KUKA KRL program: TMatriz.src, TMatriz.dat

--- TMatriz.src ---
&ACCESS RV1
DEF TMatriz()
;FOLD PALLET 1
;FOLD Pallet 1 - Produto 9Aero
;FOLD LAYER 1: PLACE 1 ate 2
;FOLD PLACE 1
;FOLD PROPRIEDADES
MatrizPontos[Pallet_1,Prdt_9Aero,1].NumCaixas = 4
MatrizPontos[Pallet_1,Prdt_9Aero,1].PickOp = 3
MatrizPontos[Pallet_1,Prdt_9Aero,1].ConfGarraOp = 3
MatrizPontos[Pallet_1,Prdt_9Aero,1].FechaGarraOp = 0
MatrizPontos[Pallet_1,Prdt_9Aero,1].AbreGarraOp = 0
MatrizPontos[Pallet_1,Prdt_9Aero,1].SensoresCaixa = 123456
MatrizPontos[Pallet_1,Prdt_9Aero,1].TravaGarra = False
MatrizPontos[Pallet_1,Prdt_9Aero,1].SkipGoHome = False
MatrizPontos[Pallet_1,Prdt_9Aero,1].SkipSobeRelAtual = False
MatrizPontos[Pallet_1,Prdt_9Aero,1].XApp1Place=P1_9Aero_1_App1
MatrizPontos[Pallet_1,Prdt_9Aero,1].XApp2Place=P1_9Aero_1_App2
MatrizPontos[Pallet_1,Prdt_9Aero,1].XPlace=P1_9Aero_1_Place
;ENDFOLD
;FOLD OffsetPlace
MatrizPontos[Pallet_1,Prdt_9Aero,1].OffsetPlace.X=0
MatrizPontos[Pallet_1,Prdt_9Aero,1].OffsetPlace.Y=0
MatrizPontos[Pallet_1,Prdt_9Aero,1].OffsetPlace.Z=0
MatrizPontos[Pallet_1,Prdt_9Aero,1].OffsetPlace.A=0
MatrizPontos[Pallet_1,Prdt_9Aero,1].OffsetPlace.B=0
MatrizPontos[Pallet_1,Prdt_9Aero,1].OffsetPlace.C=0
;ENDFOLD
;ENDFOLD

;FOLD PLACE 2
;FOLD PROPRIEDADES
MatrizPontos[Pallet_1,Prdt_9Aero,2].NumCaixas = 4
MatrizPontos[Pallet_1,Prdt_9Aero,2].PickOp = 3
MatrizPontos[Pallet_1,Prdt_9Aero,2].ConfGarraOp = 3
MatrizPontos[Pallet_1,Prdt_9Aero,2].FechaGarraOp = 0
MatrizPontos[Pallet_1,Prdt_9Aero,2].AbreGarraOp = 0
MatrizPontos[Pallet_1,Prdt_9Aero,2].SensoresCaixa = 123456
MatrizPontos[Pallet_1,Prdt_9Aero,2].TravaGarra = False
MatrizPontos[Pallet_1,Prdt_9Aero,2].SkipGoHome = False
MatrizPontos[Pallet_1,Prdt_9Aero,2].SkipSobeRelAtual = False
MatrizPontos[Pallet_1,Prdt_9Aero,2].XApp1Place=P1_9Aero_2_App1
MatrizPontos[Pallet_1,Prdt_9Aero,2].XApp2Place=P1_9Aero_2_App2
MatrizPontos[Pallet_1,Prdt_9Aero,2].XPlace=P1_9Aero_2_Place
;ENDFOLD
;FOLD OffsetPlace
MatrizPontos[Pallet_1,Prdt_9Aero,2].OffsetPlace.X=0
MatrizPontos[Pallet_1,Prdt_9Aero,2].OffsetPlace.Y=0
MatrizPontos[Pallet_1,Prdt_9Aero,2].OffsetPlace.Z=0
MatrizPontos[Pallet_1,Prdt_9Aero,2].OffsetPlace.A=0
MatrizPontos[Pallet_1,Prdt_9Aero,2].OffsetPlace.B=0
MatrizPontos[Pallet_1,Prdt_9Aero,2].OffsetPlace.C=0
;ENDFOLD
;ENDFOLD

;ENDFOLD
;ENDFOLD

;FOLD Pallet 1 - Produto 5Aero
;FOLD LAYER 1: PLACE 1 ate 3
;FOLD PLACE 1
;FOLD PROPRIEDADES
MatrizPontos[Pallet_1,Prdt_5Aero,1].NumCaixas = 3
MatrizPontos[Pallet_1,Prdt_5Aero,1].PickOp = 1
MatrizPontos[Pallet_1,Prdt_5Aero,1].ConfGarraOp = 0
MatrizPontos[Pallet_1,Prdt_5Aero,1].FechaGarraOp = 0
MatrizPontos[Pallet_1,Prdt_5Aero,1].AbreGarraOp = 0
MatrizPontos[Pallet_1,Prdt_5Aero,1].SensoresCaixa = 12345
MatrizPontos[Pallet_1,Prdt_5Aero,1].TravaGarra = False
MatrizPontos[Pallet_1,Prdt_5Aero,1].SkipGoHome = False
MatrizPontos[Pallet_1,Prdt_5Aero,1].SkipSobeRelAtual = False
MatrizPontos[Pallet_1,Prdt_5Aero,1].XApp1Place=P1_5Aero_1_App1
MatrizPontos[Pallet_1,Prdt_5Aero,1].XApp2Place=P1_5Aero_1_App2
MatrizPontos[Pallet_1,Prdt_5Aero,1].XPlace=P1_5Aero_1_Place
;ENDFOLD
;FOLD OffsetPlace
MatrizPontos[Pallet_1,Prdt_5Aero,1].OffsetPlace.X=0
MatrizPontos[Pallet_1,Prdt_5Aero,1].OffsetPlace.Y=0
MatrizPontos[Pallet_1,Prdt_5Aero,1].OffsetPlace.Z=0
MatrizPontos[Pallet_1,Prdt_5Aero,1].OffsetPlace.A=0
MatrizPontos[Pallet_1,Prdt_5Aero,1].OffsetPlace.B=0
MatrizPontos[Pallet_1,Prdt_5Aero,1].OffsetPlace.C=0
;ENDFOLD
;ENDFOLD

;FOLD PLACE 2
;FOLD PROPRIEDADES
MatrizPontos[Pallet_1,Prdt_5Aero,2].NumCaixas = 3
MatrizPontos[Pallet_1,Prdt_5Aero,2].PickOp = 1
MatrizPontos[Pallet_1,Prdt_5Aero,2].ConfGarraOp = 0
MatrizPontos[Pallet_1,Prdt_5Aero,2].FechaGarraOp = 0
MatrizPontos[Pallet_1,Prdt_5Aero,2].AbreGarraOp = 0
MatrizPontos[Pallet_1,Prdt_5Aero,2].SensoresCaixa = 12345
MatrizPontos[Pallet_1,Prdt_5Aero,2].TravaGarra = False
MatrizPontos[Pallet_1,Prdt_5Aero,2].SkipGoHome = False
MatrizPontos[Pallet_1,Prdt_5Aero,2].SkipSobeRelAtual = False
MatrizPontos[Pallet_1,Prdt_5Aero,2].XApp1Place=P1_5Aero_2_App1
MatrizPontos[Pallet_1,Prdt_5Aero,2].XApp2Place=P1_5Aero_2_App2
MatrizPontos[Pallet_1,Prdt_5Aero,2].XPlace=P1_5Aero_2_Place
;ENDFOLD
;FOLD OffsetPlace
MatrizPontos[Pallet_1,Prdt_5Aero,2].OffsetPlace.X=0
MatrizPontos[Pallet_1,Prdt_5Aero,2].OffsetPlace.Y=0
MatrizPontos[Pallet_1,Prdt_5Aero,2].OffsetPlace.Z=0
MatrizPontos[Pallet_1,Prdt_5Aero,2].OffsetPlace.A=0
MatrizPontos[Pallet_1,Prdt_5Aero,2].OffsetPlace.B=0
MatrizPontos[Pallet_1,Prdt_5Aero,2].OffsetPlace.C=0
;ENDFOLD
;ENDFOLD

;FOLD PLACE 3
;FOLD PROPRIEDADES
MatrizPontos[Pallet_1,Prdt_5Aero,3].NumCaixas = 3
MatrizPontos[Pallet_1,Prdt_5Aero,3].PickOp = 1
MatrizPontos[Pallet_1,Prdt_5Aero,3].ConfGarraOp = 0
MatrizPontos[Pallet_1,Prdt_5Aero,3].FechaGarraOp = 0
MatrizPontos[Pallet_1,Prdt_5Aero,3].AbreGarraOp = 0
MatrizPontos[Pallet_1,Prdt_5Aero,3].SensoresCaixa = 12345
MatrizPontos[Pallet_1,Prdt_5Aero,3].TravaGarra = False
MatrizPontos[Pallet_1,Prdt_5Aero,3].SkipGoHome = False
MatrizPontos[Pallet_1,Prdt_5Aero,3].SkipSobeRelAtual = False
MatrizPontos[Pallet_1,Prdt_5Aero,3].XApp1Place=P1_5Aero_3_App1
MatrizPontos[Pallet_1,Prdt_5Aero,3].XApp2Place=P1_5Aero_3_App2
MatrizPontos[Pallet_1,Prdt_5Aero,3].XPlace=P1_5Aero_3_Place
;ENDFOLD
;FOLD OffsetPlace
MatrizPontos[Pallet_1,Prdt_5Aero,3].OffsetPlace.X=0
MatrizPontos[Pallet_1,Prdt_5Aero,3].OffsetPlace.Y=0
MatrizPontos[Pallet_1,Prdt_5Aero,3].OffsetPlace.Z=0
MatrizPontos[Pallet_1,Prdt_5Aero,3].OffsetPlace.A=0
MatrizPontos[Pallet_1,Prdt_5Aero,3].OffsetPlace.B=0
MatrizPontos[Pallet_1,Prdt_5Aero,3].OffsetPlace.C=0
;ENDFOLD
;ENDFOLD

;ENDFOLD
;ENDFOLD

;FOLD Pallet 1 - Produto 2Aero
;FOLD LAYER 1: PLACE 1 ate 3
;FOLD PLACE 1
;FOLD PROPRIEDADES
MatrizPontos[Pallet_1,Prdt_2Aero,1].NumCaixas = 4
MatrizPontos[Pallet_1,Prdt_2Aero,1].PickOp = 1
MatrizPontos[Pallet_1,Prdt_2Aero,1].ConfGarraOp = 0
MatrizPontos[Pallet_1,Prdt_2Aero,1].FechaGarraOp = 0
MatrizPontos[Pallet_1,Prdt_2Aero,1].AbreGarraOp = 0
MatrizPontos[Pallet_1,Prdt_2Aero,1].SensoresCaixa = 123456
MatrizPontos[Pallet_1,Prdt_2Aero,1].TravaGarra = False
MatrizPontos[Pallet_1,Prdt_2Aero,1].SkipGoHome = False
MatrizPontos[Pallet_1,Prdt_2Aero,1].SkipSobeRelAtual = False
MatrizPontos[Pallet_1,Prdt_2Aero,1].XApp1Place=P1_2Aero_1_App1
MatrizPontos[Pallet_1,Prdt_2Aero,1].XApp2Place=P1_2Aero_1_App2
MatrizPontos[Pallet_1,Prdt_2Aero,1].XPlace=P1_2Aero_1_Place
;ENDFOLD
;FOLD OffsetPlace
MatrizPontos[Pallet_1,Prdt_2Aero,1].OffsetPlace.X=0
MatrizPontos[Pallet_1,Prdt_2Aero,1].OffsetPlace.Y=0
MatrizPontos[Pallet_1,Prdt_2Aero,1].OffsetPlace.Z=0
MatrizPontos[Pallet_1,Prdt_2Aero,1].OffsetPlace.A=0
MatrizPontos[Pallet_1,Prdt_2Aero,1].OffsetPlace.B=0
MatrizPontos[Pallet_1,Prdt_2Aero,1].OffsetPlace.C=0
;ENDFOLD
;ENDFOLD

;FOLD PLACE 2
;FOLD PROPRIEDADES
MatrizPontos[Pallet_1,Prdt_2Aero,2].NumCaixas = 4
MatrizPontos[Pallet_1,Prdt_2Aero,2].PickOp = 1
MatrizPontos[Pallet_1,Prdt_2Aero,2].ConfGarraOp = 0
MatrizPontos[Pallet_1,Prdt_2Aero,2].FechaGarraOp = 0
MatrizPontos[Pallet_1,Prdt_2Aero,2].AbreGarraOp = 0
MatrizPontos[Pallet_1,Prdt_2Aero,2].SensoresCaixa = 123456
MatrizPontos[Pallet_1,Prdt_2Aero,2].TravaGarra = False
MatrizPontos[Pallet_1,Prdt_2Aero,2].SkipGoHome = False
MatrizPontos[Pallet_1,Prdt_2Aero,2].SkipSobeRelAtual = False
MatrizPontos[Pallet_1,Prdt_2Aero,2].XApp1Place=P1_2Aero_2_App1
MatrizPontos[Pallet_1,Prdt_2Aero,2].XApp2Place=P1_2Aero_2_App2
MatrizPontos[Pallet_1,Prdt_2Aero,2].XPlace=P1_2Aero_2_Place
;ENDFOLD
;FOLD OffsetPlace
MatrizPontos[Pallet_1,Prdt_2Aero,2].OffsetPlace.X=0
MatrizPontos[Pallet_1,Prdt_2Aero,2].OffsetPlace.Y=0
MatrizPontos[Pallet_1,Prdt_2Aero,2].OffsetPlace.Z=0
MatrizPontos[Pallet_1,Prdt_2Aero,2].OffsetPlace.A=0
MatrizPontos[Pallet_1,Prdt_2Aero,2].OffsetPlace.B=0
MatrizPontos[Pallet_1,Prdt_2Aero,2].OffsetPlace.C=0
;ENDFOLD
;ENDFOLD

;FOLD PLACE 3
;FOLD PROPRIEDADES
MatrizPontos[Pallet_1,Prdt_2Aero,3].NumCaixas = 4
MatrizPontos[Pallet_1,Prdt_2Aero,3].PickOp = 1
MatrizPontos[Pallet_1,Prdt_2Aero,3].ConfGarraOp = 0
MatrizPontos[Pallet_1,Prdt_2Aero,3].FechaGarraOp = 0
MatrizPontos[Pallet_1,Prdt_2Aero,3].AbreGarraOp = 0
MatrizPontos[Pallet_1,Prdt_2Aero,3].SensoresCaixa = 123456
MatrizPontos[Pallet_1,Prdt_2Aero,3].TravaGarra = False
MatrizPontos[Pallet_1,Prdt_2Aero,3].SkipGoHome = False
MatrizPontos[Pallet_1,Prdt_2Aero,3].SkipSobeRelAtual = False
MatrizPontos[Pallet_1,Prdt_2Aero,3].XApp1Place=P1_2Aero_3_App1
MatrizPontos[Pallet_1,Prdt_2Aero,3].XApp2Place=P1_2Aero_3_App2
MatrizPontos[Pallet_1,Prdt_2Aero,3].XPlace=P1_2Aero_3_Place
;ENDFOLD
;FOLD OffsetPlace
MatrizPontos[Pallet_1,Prdt_2Aero,3].OffsetPlace.X=0
MatrizPontos[Pallet_1,Prdt_2Aero,3].OffsetPlace.Y=0
MatrizPontos[Pallet_1,Prdt_2Aero,3].OffsetPlace.Z=0
MatrizPontos[Pallet_1,Prdt_2Aero,3].OffsetPlace.A=0
MatrizPontos[Pallet_1,Prdt_2Aero,3].OffsetPlace.B=0
MatrizPontos[Pallet_1,Prdt_2Aero,3].OffsetPlace.C=0
;ENDFOLD
;ENDFOLD

;ENDFOLD
;ENDFOLD

;FOLD Pallet 1 - Produto 11CoffeCrisp
;FOLD LAYER 1: PLACE 1 ate 3
;FOLD PLACE 1
;FOLD PROPRIEDADES
MatrizPontos[Pallet_1,Prdt_11CoffeCrisp,1].NumCaixas = 3
MatrizPontos[Pallet_1,Prdt_11CoffeCrisp,1].PickOp = 1
MatrizPontos[Pallet_1,Prdt_11CoffeCrisp,1].ConfGarraOp = 0
MatrizPontos[Pallet_1,Prdt_11CoffeCrisp,1].FechaGarraOp = 0
MatrizPontos[Pallet_1,Prdt_11CoffeCrisp,1].AbreGarraOp = 0
MatrizPontos[Pallet_1,Prdt_11CoffeCrisp,1].SensoresCaixa = 12345
MatrizPontos[Pallet_1,Prdt_11CoffeCrisp,1].TravaGarra = False
MatrizPontos[Pallet_1,Prdt_11CoffeCrisp,1].SkipGoHome = False
MatrizPontos[Pallet_1,Prdt_11CoffeCrisp,1].SkipSobeRelAtual = False
MatrizPontos[Pallet_1,Prdt_11CoffeCrisp,1].XApp1Place=P1_11CoffeCrisp_1_App1
MatrizPontos[Pallet_1,Prdt_11CoffeCrisp,1].XApp2Place=P1_11CoffeCrisp_1_App2
MatrizPontos[Pallet_1,Prdt_11CoffeCrisp,1].XPlace=P1_11CoffeCrisp_1_Place
;ENDFOLD
;FOLD OffsetPlace
MatrizPontos[Pallet_1,Prdt_11CoffeCrisp,1].OffsetPlace.X=0
MatrizPontos[Pallet_1,Prdt_11CoffeCrisp,1].OffsetPlace.Y=0
MatrizPontos[Pallet_1,Prdt_11CoffeCrisp,1].OffsetPlace.Z=0
MatrizPontos[Pallet_1,Prdt_11CoffeCrisp,1].OffsetPlace.A=0
MatrizPontos[Pallet_1,Prdt_11CoffeCrisp,1].OffsetPlace.B=0
MatrizPontos[Pallet_1,Prdt_11CoffeCrisp,1].OffsetPlace.C=0
;ENDFOLD
;ENDFOLD

;FOLD PLACE 2
;FOLD PROPRIEDADES
MatrizPontos[Pallet_1,Prdt_11CoffeCrisp,2].NumCaixas = 3
MatrizPontos[Pallet_1,Prdt_11CoffeCrisp,2].PickOp = 1
MatrizPontos[Pallet_1,Prdt_11CoffeCrisp,2].ConfGarraOp = 0
MatrizPontos[Pallet_1,Prdt_11CoffeCrisp,2].FechaGarraOp = 0
MatrizPontos[Pallet_1,Prdt_11CoffeCrisp,2].AbreGarraOp = 0
MatrizPontos[Pallet_1,Prdt_11CoffeCrisp,2].SensoresCaixa = 12345
MatrizPontos[Pallet_1,Prdt_11CoffeCrisp,2].TravaGarra = False
MatrizPontos[Pallet_1,Prdt_11CoffeCrisp,2].SkipGoHome = False
MatrizPontos[Pallet_1,Prdt_11CoffeCrisp,2].SkipSobeRelAtual = False
MatrizPontos[Pallet_1,Prdt_11CoffeCrisp,2].XApp1Place=P1_11CoffeCrisp_2_App1
MatrizPontos[Pallet_1,Prdt_11CoffeCrisp,2].XApp2Place=P1_11CoffeCrisp_2_App2
MatrizPontos[Pallet_1,Prdt_11CoffeCrisp,2].XPlace=P1_11CoffeCrisp_2_Place
;ENDFOLD
;FOLD OffsetPlace
MatrizPontos[Pallet_1,Prdt_11CoffeCrisp,2].OffsetPlace.X=0
MatrizPontos[Pallet_1,Prdt_11CoffeCrisp,2].OffsetPlace.Y=0
MatrizPontos[Pallet_1,Prdt_11CoffeCrisp,2].OffsetPlace.Z=0
MatrizPontos[Pallet_1,Prdt_11CoffeCrisp,2].OffsetPlace.A=0
MatrizPontos[Pallet_1,Prdt_11CoffeCrisp,2].OffsetPlace.B=0
MatrizPontos[Pallet_1,Prdt_11CoffeCrisp,2].OffsetPlace.C=0
;ENDFOLD
;ENDFOLD

;FOLD PLACE 3
;FOLD PROPRIEDADES
MatrizPontos[Pallet_1,Prdt_11CoffeCrisp,3].NumCaixas = 3
MatrizPontos[Pallet_1,Prdt_11CoffeCrisp,3].PickOp = 1
MatrizPontos[Pallet_1,Prdt_11CoffeCrisp,3].ConfGarraOp = 0
MatrizPontos[Pallet_1,Prdt_11CoffeCrisp,3].FechaGarraOp = 0
MatrizPontos[Pallet_1,Prdt_11CoffeCrisp,3].AbreGarraOp = 0
MatrizPontos[Pallet_1,Prdt_11CoffeCrisp,3].SensoresCaixa = 12345
MatrizPontos[Pallet_1,Prdt_11CoffeCrisp,3].TravaGarra = False
MatrizPontos[Pallet_1,Prdt_11CoffeCrisp,3].SkipGoHome = False
MatrizPontos[Pallet_1,Prdt_11CoffeCrisp,3].SkipSobeRelAtual = False
MatrizPontos[Pallet_1,Prdt_11CoffeCrisp,3].XApp1Place=P1_11CoffeCrisp_3_App1
MatrizPontos[Pallet_1,Prdt_11CoffeCrisp,3].XApp2Place=P1_11CoffeCrisp_3_App2
MatrizPontos[Pallet_1,Prdt_11CoffeCrisp,3].XPlace=P1_11CoffeCrisp_3_Place
;ENDFOLD
;FOLD OffsetPlace
MatrizPontos[Pallet_1,Prdt_11CoffeCrisp,3].OffsetPlace.X=0
MatrizPontos[Pallet_1,Prdt_11CoffeCrisp,3].OffsetPlace.Y=0
MatrizPontos[Pallet_1,Prdt_11CoffeCrisp,3].OffsetPlace.Z=0
MatrizPontos[Pallet_1,Prdt_11CoffeCrisp,3].OffsetPlace.A=0
MatrizPontos[Pallet_1,Prdt_11CoffeCrisp,3].OffsetPlace.B=0
MatrizPontos[Pallet_1,Prdt_11CoffeCrisp,3].OffsetPlace.C=0
;ENDFOLD
;ENDFOLD

;ENDFOLD
;ENDFOLD

;FOLD Pallet 1 - Produto 17KitKat
;FOLD LAYER 1: PLACE 1 ate 4
;FOLD PLACE 1
;FOLD PROPRIEDADES
MatrizPontos[Pallet_1,Prdt_17KitKat,1].NumCaixas = 3
MatrizPontos[Pallet_1,Prdt_17KitKat,1].PickOp = 1
MatrizPontos[Pallet_1,Prdt_17KitKat,1].ConfGarraOp = 0
MatrizPontos[Pallet_1,Prdt_17KitKat,1].FechaGarraOp = 0
MatrizPontos[Pallet_1,Prdt_17KitKat,1].AbreGarraOp = 0
MatrizPontos[Pallet_1,Prdt_17KitKat,1].SensoresCaixa = 1234
MatrizPontos[Pallet_1,Prdt_17KitKat,1].TravaGarra = False
MatrizPontos[Pallet_1,Prdt_17KitKat,1].SkipGoHome = False
MatrizPontos[Pallet_1,Prdt_17KitKat,1].SkipSobeRelAtual = False
MatrizPontos[Pallet_1,Prdt_17KitKat,1].XApp1Place=P1_17KitKat_1_App1
MatrizPontos[Pallet_1,Prdt_17KitKat,1].XApp2Place=P1_17KitKat_1_App2
MatrizPontos[Pallet_1,Prdt_17KitKat,1].XPlace=P1_17KitKat_1_Place
;ENDFOLD
;FOLD OffsetPlace
MatrizPontos[Pallet_1,Prdt_17KitKat,1].OffsetPlace.X=0
MatrizPontos[Pallet_1,Prdt_17KitKat,1].OffsetPlace.Y=0
MatrizPontos[Pallet_1,Prdt_17KitKat,1].OffsetPlace.Z=0
MatrizPontos[Pallet_1,Prdt_17KitKat,1].OffsetPlace.A=0
MatrizPontos[Pallet_1,Prdt_17KitKat,1].OffsetPlace.B=0
MatrizPontos[Pallet_1,Prdt_17KitKat,1].OffsetPlace.C=0
;ENDFOLD
;ENDFOLD

;FOLD PLACE 2
;FOLD PROPRIEDADES
MatrizPontos[Pallet_1,Prdt_17KitKat,2].NumCaixas = 3
MatrizPontos[Pallet_1,Prdt_17KitKat,2].PickOp = 1
MatrizPontos[Pallet_1,Prdt_17KitKat,2].ConfGarraOp = 0
MatrizPontos[Pallet_1,Prdt_17KitKat,2].FechaGarraOp = 0
MatrizPontos[Pallet_1,Prdt_17KitKat,2].AbreGarraOp = 0
MatrizPontos[Pallet_1,Prdt_17KitKat,2].SensoresCaixa = 1234
MatrizPontos[Pallet_1,Prdt_17KitKat,2].TravaGarra = False
MatrizPontos[Pallet_1,Prdt_17KitKat,2].SkipGoHome = False
MatrizPontos[Pallet_1,Prdt_17KitKat,2].SkipSobeRelAtual = False
MatrizPontos[Pallet_1,Prdt_17KitKat,2].XApp1Place=P1_17KitKat_2_App1
MatrizPontos[Pallet_1,Prdt_17KitKat,2].XApp2Place=P1_17KitKat_2_App2
MatrizPontos[Pallet_1,Prdt_17KitKat,2].XPlace=P1_17KitKat_2_Place
;ENDFOLD
;FOLD OffsetPlace
MatrizPontos[Pallet_1,Prdt_17KitKat,2].OffsetPlace.X=0
MatrizPontos[Pallet_1,Prdt_17KitKat,2].OffsetPlace.Y=0
MatrizPontos[Pallet_1,Prdt_17KitKat,2].OffsetPlace.Z=0
MatrizPontos[Pallet_1,Prdt_17KitKat,2].OffsetPlace.A=0
MatrizPontos[Pallet_1,Prdt_17KitKat,2].OffsetPlace.B=0
MatrizPontos[Pallet_1,Prdt_17KitKat,2].OffsetPlace.C=0
;ENDFOLD
;ENDFOLD

;FOLD PLACE 3
;FOLD PROPRIEDADES
MatrizPontos[Pallet_1,Prdt_17KitKat,3].NumCaixas = 3
MatrizPontos[Pallet_1,Prdt_17KitKat,3].PickOp = 1
MatrizPontos[Pallet_1,Prdt_17KitKat,3].ConfGarraOp = 0
MatrizPontos[Pallet_1,Prdt_17KitKat,3].FechaGarraOp = 0
MatrizPontos[Pallet_1,Prdt_17KitKat,3].AbreGarraOp = 0
MatrizPontos[Pallet_1,Prdt_17KitKat,3].SensoresCaixa = 1234
MatrizPontos[Pallet_1,Prdt_17KitKat,3].TravaGarra = False
MatrizPontos[Pallet_1,Prdt_17KitKat,3].SkipGoHome = False
MatrizPontos[Pallet_1,Prdt_17KitKat,3].SkipSobeRelAtual = False
MatrizPontos[Pallet_1,Prdt_17KitKat,3].XApp1Place=P1_17KitKat_3_App1
MatrizPontos[Pallet_1,Prdt_17KitKat,3].XApp2Place=P1_17KitKat_3_App2
MatrizPontos[Pallet_1,Prdt_17KitKat,3].XPlace=P1_17KitKat_3_Place
;ENDFOLD
;FOLD OffsetPlace
MatrizPontos[Pallet_1,Prdt_17KitKat,3].OffsetPlace.X=0
MatrizPontos[Pallet_1,Prdt_17KitKat,3].OffsetPlace.Y=0
MatrizPontos[Pallet_1,Prdt_17KitKat,3].OffsetPlace.Z=0
MatrizPontos[Pallet_1,Prdt_17KitKat,3].OffsetPlace.A=0
MatrizPontos[Pallet_1,Prdt_17KitKat,3].OffsetPlace.B=0
MatrizPontos[Pallet_1,Prdt_17KitKat,3].OffsetPlace.C=0
;ENDFOLD
;ENDFOLD

;FOLD PLACE 4
;FOLD PROPRIEDADES
MatrizPontos[Pallet_1,Prdt_17KitKat,4].NumCaixas = 3
MatrizPontos[Pallet_1,Prdt_17KitKat,4].PickOp = 1
MatrizPontos[Pallet_1,Prdt_17KitKat,4].ConfGarraOp = 0
MatrizPontos[Pallet_1,Prdt_17KitKat,4].FechaGarraOp = 0
MatrizPontos[Pallet_1,Prdt_17KitKat,4].AbreGarraOp = 0
MatrizPontos[Pallet_1,Prdt_17KitKat,4].SensoresCaixa = 1234
MatrizPontos[Pallet_1,Prdt_17KitKat,4].TravaGarra = False
MatrizPontos[Pallet_1,Prdt_17KitKat,4].SkipGoHome = False
MatrizPontos[Pallet_1,Prdt_17KitKat,4].SkipSobeRelAtual = False
MatrizPontos[Pallet_1,Prdt_17KitKat,4].XApp1Place=P1_17KitKat_4_App1
MatrizPontos[Pallet_1,Prdt_17KitKat,4].XApp2Place=P1_17KitKat_4_App2
MatrizPontos[Pallet_1,Prdt_17KitKat,4].XPlace=P1_17KitKat_4_Place
;ENDFOLD
;FOLD OffsetPlace
MatrizPontos[Pallet_1,Prdt_17KitKat,4].OffsetPlace.X=0
MatrizPontos[Pallet_1,Prdt_17KitKat,4].OffsetPlace.Y=0
MatrizPontos[Pallet_1,Prdt_17KitKat,4].OffsetPlace.Z=0
MatrizPontos[Pallet_1,Prdt_17KitKat,4].OffsetPlace.A=0
MatrizPontos[Pallet_1,Prdt_17KitKat,4].OffsetPlace.B=0
MatrizPontos[Pallet_1,Prdt_17KitKat,4].OffsetPlace.C=0
;ENDFOLD
;ENDFOLD

;ENDFOLD
;ENDFOLD

;FOLD Pallet 1 - Produto 19KitKat
;FOLD LAYER 1: PLACE 1 ate 6
;FOLD PLACE 1
;FOLD PROPRIEDADES
MatrizPontos[Pallet_1,Prdt_19KitKat,1].NumCaixas = 1
MatrizPontos[Pallet_1,Prdt_19KitKat,1].PickOp = 6
MatrizPontos[Pallet_1,Prdt_19KitKat,1].ConfGarraOp = 0
MatrizPontos[Pallet_1,Prdt_19KitKat,1].FechaGarraOp = 0
MatrizPontos[Pallet_1,Prdt_19KitKat,1].AbreGarraOp = 0
MatrizPontos[Pallet_1,Prdt_19KitKat,1].SensoresCaixa = 6
MatrizPontos[Pallet_1,Prdt_19KitKat,1].TravaGarra = False
MatrizPontos[Pallet_1,Prdt_19KitKat,1].SkipGoHome = False
MatrizPontos[Pallet_1,Prdt_19KitKat,1].SkipSobeRelAtual = False
MatrizPontos[Pallet_1,Prdt_19KitKat,1].XApp1Place=P1_19KitKat_1_App1
MatrizPontos[Pallet_1,Prdt_19KitKat,1].XApp2Place=P1_19KitKat_1_App2
MatrizPontos[Pallet_1,Prdt_19KitKat,1].XPlace=P1_19KitKat_1_Place
;ENDFOLD
;FOLD OffsetPlace
MatrizPontos[Pallet_1,Prdt_19KitKat,1].OffsetPlace.X=0
MatrizPontos[Pallet_1,Prdt_19KitKat,1].OffsetPlace.Y=0
MatrizPontos[Pallet_1,Prdt_19KitKat,1].OffsetPlace.Z=0
MatrizPontos[Pallet_1,Prdt_19KitKat,1].OffsetPlace.A=0
MatrizPontos[Pallet_1,Prdt_19KitKat,1].OffsetPlace.B=0
MatrizPontos[Pallet_1,Prdt_19KitKat,1].OffsetPlace.C=0
;ENDFOLD
;ENDFOLD

;FOLD PLACE 2
;FOLD PROPRIEDADES
MatrizPontos[Pallet_1,Prdt_19KitKat,2].NumCaixas = 1
MatrizPontos[Pallet_1,Prdt_19KitKat,2].PickOp = 6
MatrizPontos[Pallet_1,Prdt_19KitKat,2].ConfGarraOp = 0
MatrizPontos[Pallet_1,Prdt_19KitKat,2].FechaGarraOp = 0
MatrizPontos[Pallet_1,Prdt_19KitKat,2].AbreGarraOp = 0
MatrizPontos[Pallet_1,Prdt_19KitKat,2].SensoresCaixa = 6
MatrizPontos[Pallet_1,Prdt_19KitKat,2].TravaGarra = False
MatrizPontos[Pallet_1,Prdt_19KitKat,2].SkipGoHome = False
MatrizPontos[Pallet_1,Prdt_19KitKat,2].SkipSobeRelAtual = False
MatrizPontos[Pallet_1,Prdt_19KitKat,2].XApp1Place=P1_19KitKat_2_App1
MatrizPontos[Pallet_1,Prdt_19KitKat,2].XApp2Place=P1_19KitKat_2_App2
MatrizPontos[Pallet_1,Prdt_19KitKat,2].XPlace=P1_19KitKat_2_Place
;ENDFOLD
;FOLD OffsetPlace
MatrizPontos[Pallet_1,Prdt_19KitKat,2].OffsetPlace.X=0
MatrizPontos[Pallet_1,Prdt_19KitKat,2].OffsetPlace.Y=0
MatrizPontos[Pallet_1,Prdt_19KitKat,2].OffsetPlace.Z=0
MatrizPontos[Pallet_1,Prdt_19KitKat,2].OffsetPlace.A=0
MatrizPontos[Pallet_1,Prdt_19KitKat,2].OffsetPlace.B=0
MatrizPontos[Pallet_1,Prdt_19KitKat,2].OffsetPlace.C=0
;ENDFOLD
;ENDFOLD

;FOLD PLACE 3
;FOLD PROPRIEDADES
MatrizPontos[Pallet_1,Prdt_19KitKat,3].NumCaixas = 1
MatrizPontos[Pallet_1,Prdt_19KitKat,3].PickOp = 6
MatrizPontos[Pallet_1,Prdt_19KitKat,3].ConfGarraOp = 0
MatrizPontos[Pallet_1,Prdt_19KitKat,3].FechaGarraOp = 0
MatrizPontos[Pallet_1,Prdt_19KitKat,3].AbreGarraOp = 0
MatrizPontos[Pallet_1,Prdt_19KitKat,3].SensoresCaixa = 6
MatrizPontos[Pallet_1,Prdt_19KitKat,3].TravaGarra = False
MatrizPontos[Pallet_1,Prdt_19KitKat,3].SkipGoHome = False
MatrizPontos[Pallet_1,Prdt_19KitKat,3].SkipSobeRelAtual = False
MatrizPontos[Pallet_1,Prdt_19KitKat,3].XApp1Place=P1_19KitKat_3_App1
MatrizPontos[Pallet_1,Prdt_19KitKat,3].XApp2Place=P1_19KitKat_3_App2
MatrizPontos[Pallet_1,Prdt_19KitKat,3].XPlace=P1_19KitKat_3_Place
;ENDFOLD
;FOLD OffsetPlace
MatrizPontos[Pallet_1,Prdt_19KitKat,3].OffsetPlace.X=0
MatrizPontos[Pallet_1,Prdt_19KitKat,3].OffsetPlace.Y=0
MatrizPontos[Pallet_1,Prdt_19KitKat,3].OffsetPlace.Z=0
MatrizPontos[Pallet_1,Prdt_19KitKat,3].OffsetPlace.A=0
MatrizPontos[Pallet_1,Prdt_19KitKat,3].OffsetPlace.B=0
MatrizPontos[Pallet_1,Prdt_19KitKat,3].OffsetPlace.C=0
;ENDFOLD
;ENDFOLD

;FOLD PLACE 4
;FOLD PROPRIEDADES
MatrizPontos[Pallet_1,Prdt_19KitKat,4].NumCaixas = 4
MatrizPontos[Pallet_1,Prdt_19KitKat,4].PickOp = 1
MatrizPontos[Pallet_1,Prdt_19KitKat,4].ConfGarraOp = 0
MatrizPontos[Pallet_1,Prdt_19KitKat,4].FechaGarraOp = 0
MatrizPontos[Pallet_1,Prdt_19KitKat,4].AbreGarraOp = 0
MatrizPontos[Pallet_1,Prdt_19KitKat,4].SensoresCaixa = 12345
MatrizPontos[Pallet_1,Prdt_19KitKat,4].TravaGarra = False
MatrizPontos[Pallet_1,Prdt_19KitKat,4].SkipGoHome = False
MatrizPontos[Pallet_1,Prdt_19KitKat,4].SkipSobeRelAtual = False
MatrizPontos[Pallet_1,Prdt_19KitKat,4].XApp1Place=P1_19KitKat_4_App1
MatrizPontos[Pallet_1,Prdt_19KitKat,4].XApp2Place=P1_19KitKat_4_App2
MatrizPontos[Pallet_1,Prdt_19KitKat,4].XPlace=P1_19KitKat_4_Place
;ENDFOLD
;FOLD OffsetPlace
MatrizPontos[Pallet_1,Prdt_19KitKat,4].OffsetPlace.X=0
MatrizPontos[Pallet_1,Prdt_19KitKat,4].OffsetPlace.Y=0
MatrizPontos[Pallet_1,Prdt_19KitKat,4].OffsetPlace.Z=0
MatrizPontos[Pallet_1,Prdt_19KitKat,4].OffsetPlace.A=0
MatrizPontos[Pallet_1,Prdt_19KitKat,4].OffsetPlace.B=0
MatrizPontos[Pallet_1,Prdt_19KitKat,4].OffsetPlace.C=0
;ENDFOLD
;ENDFOLD

;FOLD PLACE 5
;FOLD PROPRIEDADES
MatrizPontos[Pallet_1,Prdt_19KitKat,5].NumCaixas = 4
MatrizPontos[Pallet_1,Prdt_19KitKat,5].PickOp = 1
MatrizPontos[Pallet_1,Prdt_19KitKat,5].ConfGarraOp = 0
MatrizPontos[Pallet_1,Prdt_19KitKat,5].FechaGarraOp = 0
MatrizPontos[Pallet_1,Prdt_19KitKat,5].AbreGarraOp = 0
MatrizPontos[Pallet_1,Prdt_19KitKat,5].SensoresCaixa = 12345
MatrizPontos[Pallet_1,Prdt_19KitKat,5].TravaGarra = False
MatrizPontos[Pallet_1,Prdt_19KitKat,5].SkipGoHome = False
MatrizPontos[Pallet_1,Prdt_19KitKat,5].SkipSobeRelAtual = False
MatrizPontos[Pallet_1,Prdt_19KitKat,5].XApp1Place=P1_19KitKat_5_App1
MatrizPontos[Pallet_1,Prdt_19KitKat,5].XApp2Place=P1_19KitKat_5_App2
MatrizPontos[Pallet_1,Prdt_19KitKat,5].XPlace=P1_19KitKat_5_Place
;ENDFOLD
;FOLD OffsetPlace
MatrizPontos[Pallet_1,Prdt_19KitKat,5].OffsetPlace.X=0
MatrizPontos[Pallet_1,Prdt_19KitKat,5].OffsetPlace.Y=0
MatrizPontos[Pallet_1,Prdt_19KitKat,5].OffsetPlace.Z=0
MatrizPontos[Pallet_1,Prdt_19KitKat,5].OffsetPlace.A=0
MatrizPontos[Pallet_1,Prdt_19KitKat,5].OffsetPlace.B=0
MatrizPontos[Pallet_1,Prdt_19KitKat,5].OffsetPlace.C=0
;ENDFOLD
;ENDFOLD

;FOLD PLACE 6
;FOLD PROPRIEDADES
MatrizPontos[Pallet_1,Prdt_19KitKat,6].NumCaixas = 4
MatrizPontos[Pallet_1,Prdt_19KitKat,6].PickOp = 1
MatrizPontos[Pallet_1,Prdt_19KitKat,6].ConfGarraOp = 0
MatrizPontos[Pallet_1,Prdt_19KitKat,6].FechaGarraOp = 0
MatrizPontos[Pallet_1,Prdt_19KitKat,6].AbreGarraOp = 0
MatrizPontos[Pallet_1,Prdt_19KitKat,6].SensoresCaixa = 12345
MatrizPontos[Pallet_1,Prdt_19KitKat,6].TravaGarra = False
MatrizPontos[Pallet_1,Prdt_19KitKat,6].SkipGoHome = False
MatrizPontos[Pallet_1,Prdt_19KitKat,6].SkipSobeRelAtual = False
MatrizPontos[Pallet_1,Prdt_19KitKat,6].XApp1Place=P1_19KitKat_6_App1
MatrizPontos[Pallet_1,Prdt_19KitKat,6].XApp2Place=P1_19KitKat_6_App2
MatrizPontos[Pallet_1,Prdt_19KitKat,6].XPlace=P1_19KitKat_6_Place
;ENDFOLD
;FOLD OffsetPlace
MatrizPontos[Pallet_1,Prdt_19KitKat,6].OffsetPlace.X=0
MatrizPontos[Pallet_1,Prdt_19KitKat,6].OffsetPlace.Y=0
MatrizPontos[Pallet_1,Prdt_19KitKat,6].OffsetPlace.Z=0
MatrizPontos[Pallet_1,Prdt_19KitKat,6].OffsetPlace.A=0
MatrizPontos[Pallet_1,Prdt_19KitKat,6].OffsetPlace.B=0
MatrizPontos[Pallet_1,Prdt_19KitKat,6].OffsetPlace.C=0
;ENDFOLD
;ENDFOLD

;ENDFOLD
;FOLD LAYER 2: PLACE 7 ate 12
;FOLD PLACE 7
;FOLD PROPRIEDADES
MatrizPontos[Pallet_1,Prdt_19KitKat,7].NumCaixas = 1
MatrizPontos[Pallet_1,Prdt_19KitKat,7].PickOp = 1
MatrizPontos[Pallet_1,Prdt_19KitKat,7].ConfGarraOp = 0
MatrizPontos[Pallet_1,Prdt_19KitKat,7].FechaGarraOp = 0
MatrizPontos[Pallet_1,Prdt_19KitKat,7].AbreGarraOp = 0
MatrizPontos[Pallet_1,Prdt_19KitKat,7].SensoresCaixa = 1
MatrizPontos[Pallet_1,Prdt_19KitKat,7].TravaGarra = False
MatrizPontos[Pallet_1,Prdt_19KitKat,7].SkipGoHome = False
MatrizPontos[Pallet_1,Prdt_19KitKat,7].SkipSobeRelAtual = False
MatrizPontos[Pallet_1,Prdt_19KitKat,7].XApp1Place=P1_19KitKat_7_App1
MatrizPontos[Pallet_1,Prdt_19KitKat,7].XApp2Place=P1_19KitKat_7_App2
MatrizPontos[Pallet_1,Prdt_19KitKat,7].XPlace=P1_19KitKat_7_Place
;ENDFOLD
;FOLD OffsetPlace
MatrizPontos[Pallet_1,Prdt_19KitKat,7].OffsetPlace.X=0
MatrizPontos[Pallet_1,Prdt_19KitKat,7].OffsetPlace.Y=0
MatrizPontos[Pallet_1,Prdt_19KitKat,7].OffsetPlace.Z=0
MatrizPontos[Pallet_1,Prdt_19KitKat,7].OffsetPlace.A=0
MatrizPontos[Pallet_1,Prdt_19KitKat,7].OffsetPlace.B=0
MatrizPontos[Pallet_1,Prdt_19KitKat,7].OffsetPlace.C=0
;ENDFOLD
;ENDFOLD

;FOLD PLACE 8
;FOLD PROPRIEDADES
MatrizPontos[Pallet_1,Prdt_19KitKat,8].NumCaixas = 1
MatrizPontos[Pallet_1,Prdt_19KitKat,8].PickOp = 1
MatrizPontos[Pallet_1,Prdt_19KitKat,8].ConfGarraOp = 0
MatrizPontos[Pallet_1,Prdt_19KitKat,8].FechaGarraOp = 0
MatrizPontos[Pallet_1,Prdt_19KitKat,8].AbreGarraOp = 0
MatrizPontos[Pallet_1,Prdt_19KitKat,8].SensoresCaixa = 1
MatrizPontos[Pallet_1,Prdt_19KitKat,8].TravaGarra = False
MatrizPontos[Pallet_1,Prdt_19KitKat,8].SkipGoHome = False
MatrizPontos[Pallet_1,Prdt_19KitKat,8].SkipSobeRelAtual = False
MatrizPontos[Pallet_1,Prdt_19KitKat,8].XApp1Place=P1_19KitKat_8_App1
MatrizPontos[Pallet_1,Prdt_19KitKat,8].XApp2Place=P1_19KitKat_8_App2
MatrizPontos[Pallet_1,Prdt_19KitKat,8].XPlace=P1_19KitKat_8_Place
;ENDFOLD
;FOLD OffsetPlace
MatrizPontos[Pallet_1,Prdt_19KitKat,8].OffsetPlace.X=0
MatrizPontos[Pallet_1,Prdt_19KitKat,8].OffsetPlace.Y=0
MatrizPontos[Pallet_1,Prdt_19KitKat,8].OffsetPlace.Z=0
MatrizPontos[Pallet_1,Prdt_19KitKat,8].OffsetPlace.A=0
MatrizPontos[Pallet_1,Prdt_19KitKat,8].OffsetPlace.B=0
MatrizPontos[Pallet_1,Prdt_19KitKat,8].OffsetPlace.C=0
;ENDFOLD
;ENDFOLD

;FOLD PLACE 9
;FOLD PROPRIEDADES
MatrizPontos[Pallet_1,Prdt_19KitKat,9].NumCaixas = 1
MatrizPontos[Pallet_1,Prdt_19KitKat,9].PickOp = 1
MatrizPontos[Pallet_1,Prdt_19KitKat,9].ConfGarraOp = 0
MatrizPontos[Pallet_1,Prdt_19KitKat,9].FechaGarraOp = 0
MatrizPontos[Pallet_1,Prdt_19KitKat,9].AbreGarraOp = 0
MatrizPontos[Pallet_1,Prdt_19KitKat,9].SensoresCaixa = 1
MatrizPontos[Pallet_1,Prdt_19KitKat,9].TravaGarra = False
MatrizPontos[Pallet_1,Prdt_19KitKat,9].SkipGoHome = False
MatrizPontos[Pallet_1,Prdt_19KitKat,9].SkipSobeRelAtual = False
MatrizPontos[Pallet_1,Prdt_19KitKat,9].XApp1Place=P1_19KitKat_9_App1
MatrizPontos[Pallet_1,Prdt_19KitKat,9].XApp2Place=P1_19KitKat_9_App2
MatrizPontos[Pallet_1,Prdt_19KitKat,9].XPlace=P1_19KitKat_9_Place
;ENDFOLD
;FOLD OffsetPlace
MatrizPontos[Pallet_1,Prdt_19KitKat,9].OffsetPlace.X=0
MatrizPontos[Pallet_1,Prdt_19KitKat,9].OffsetPlace.Y=0
MatrizPontos[Pallet_1,Prdt_19KitKat,9].OffsetPlace.Z=0
MatrizPontos[Pallet_1,Prdt_19KitKat,9].OffsetPlace.A=0
MatrizPontos[Pallet_1,Prdt_19KitKat,9].OffsetPlace.B=0
MatrizPontos[Pallet_1,Prdt_19KitKat,9].OffsetPlace.C=0
;ENDFOLD
;ENDFOLD

;FOLD PLACE 10
;FOLD PROPRIEDADES
MatrizPontos[Pallet_1,Prdt_19KitKat,10].NumCaixas = 4
MatrizPontos[Pallet_1,Prdt_19KitKat,10].PickOp = 1
MatrizPontos[Pallet_1,Prdt_19KitKat,10].ConfGarraOp = 0
MatrizPontos[Pallet_1,Prdt_19KitKat,10].FechaGarraOp = 0
MatrizPontos[Pallet_1,Prdt_19KitKat,10].AbreGarraOp = 1
MatrizPontos[Pallet_1,Prdt_19KitKat,10].SensoresCaixa = 12345
MatrizPontos[Pallet_1,Prdt_19KitKat,10].TravaGarra = True
MatrizPontos[Pallet_1,Prdt_19KitKat,10].SkipGoHome = False
MatrizPontos[Pallet_1,Prdt_19KitKat,10].SkipSobeRelAtual = False
MatrizPontos[Pallet_1,Prdt_19KitKat,10].XApp1Place=P1_19KitKat_10_App1
MatrizPontos[Pallet_1,Prdt_19KitKat,10].XApp2Place=P1_19KitKat_10_App2
MatrizPontos[Pallet_1,Prdt_19KitKat,10].XPlace=P1_19KitKat_10_Place
;ENDFOLD
;FOLD OffsetPlace
MatrizPontos[Pallet_1,Prdt_19KitKat,10].OffsetPlace.X=0
MatrizPontos[Pallet_1,Prdt_19KitKat,10].OffsetPlace.Y=0
MatrizPontos[Pallet_1,Prdt_19KitKat,10].OffsetPlace.Z=0
MatrizPontos[Pallet_1,Prdt_19KitKat,10].OffsetPlace.A=0
MatrizPontos[Pallet_1,Prdt_19KitKat,10].OffsetPlace.B=0
MatrizPontos[Pallet_1,Prdt_19KitKat,10].OffsetPlace.C=0
;ENDFOLD
;ENDFOLD

;FOLD PLACE 11
;FOLD PROPRIEDADES
MatrizPontos[Pallet_1,Prdt_19KitKat,11].NumCaixas = 4
MatrizPontos[Pallet_1,Prdt_19KitKat,11].PickOp = 1
MatrizPontos[Pallet_1,Prdt_19KitKat,11].ConfGarraOp = 0
MatrizPontos[Pallet_1,Prdt_19KitKat,11].FechaGarraOp = 0
MatrizPontos[Pallet_1,Prdt_19KitKat,11].AbreGarraOp = 1
MatrizPontos[Pallet_1,Prdt_19KitKat,11].SensoresCaixa = 12345
MatrizPontos[Pallet_1,Prdt_19KitKat,11].TravaGarra = True
MatrizPontos[Pallet_1,Prdt_19KitKat,11].SkipGoHome = False
MatrizPontos[Pallet_1,Prdt_19KitKat,11].SkipSobeRelAtual = False
MatrizPontos[Pallet_1,Prdt_19KitKat,11].XApp1Place=P1_19KitKat_11_App1
MatrizPontos[Pallet_1,Prdt_19KitKat,11].XApp2Place=P1_19KitKat_11_App2
MatrizPontos[Pallet_1,Prdt_19KitKat,11].XPlace=P1_19KitKat_11_Place
;ENDFOLD
;FOLD OffsetPlace
MatrizPontos[Pallet_1,Prdt_19KitKat,11].OffsetPlace.X=0
MatrizPontos[Pallet_1,Prdt_19KitKat,11].OffsetPlace.Y=0
MatrizPontos[Pallet_1,Prdt_19KitKat,11].OffsetPlace.Z=0
MatrizPontos[Pallet_1,Prdt_19KitKat,11].OffsetPlace.A=0
MatrizPontos[Pallet_1,Prdt_19KitKat,11].OffsetPlace.B=0
MatrizPontos[Pallet_1,Prdt_19KitKat,11].OffsetPlace.C=0
;ENDFOLD
;ENDFOLD

;FOLD PLACE 12
;FOLD PROPRIEDADES
MatrizPontos[Pallet_1,Prdt_19KitKat,12].NumCaixas = 4
MatrizPontos[Pallet_1,Prdt_19KitKat,12].PickOp = 1
MatrizPontos[Pallet_1,Prdt_19KitKat,12].ConfGarraOp = 0
MatrizPontos[Pallet_1,Prdt_19KitKat,12].FechaGarraOp = 0
MatrizPontos[Pallet_1,Prdt_19KitKat,12].AbreGarraOp = 1
MatrizPontos[Pallet_1,Prdt_19KitKat,12].SensoresCaixa = 12345
MatrizPontos[Pallet_1,Prdt_19KitKat,12].TravaGarra = True
MatrizPontos[Pallet_1,Prdt_19KitKat,12].SkipGoHome = False
MatrizPontos[Pallet_1,Prdt_19KitKat,12].SkipSobeRelAtual = False
MatrizPontos[Pallet_1,Prdt_19KitKat,12].XApp1Place=P1_19KitKat_12_App1
MatrizPontos[Pallet_1,Prdt_19KitKat,12].XApp2Place=P1_19KitKat_12_App2
MatrizPontos[Pallet_1,Prdt_19KitKat,12].XPlace=P1_19KitKat_12_Place
;ENDFOLD
;FOLD OffsetPlace
MatrizPontos[Pallet_1,Prdt_19KitKat,12].OffsetPlace.X=0
MatrizPontos[Pallet_1,Prdt_19KitKat,12].OffsetPlace.Y=0
MatrizPontos[Pallet_1,Prdt_19KitKat,12].OffsetPlace.Z=0
MatrizPontos[Pallet_1,Prdt_19KitKat,12].OffsetPlace.A=0
MatrizPontos[Pallet_1,Prdt_19KitKat,12].OffsetPlace.B=0
MatrizPontos[Pallet_1,Prdt_19KitKat,12].OffsetPlace.C=0
;ENDFOLD
;ENDFOLD

;ENDFOLD
;ENDFOLD

;FOLD Pallet 1 - Produto 20KitKat
;FOLD LAYER 1: PLACE 1 ate 3
;FOLD PLACE 1
;FOLD PROPRIEDADES
MatrizPontos[Pallet_1,Prdt_20KitKat,1].NumCaixas = 4
MatrizPontos[Pallet_1,Prdt_20KitKat,1].PickOp = 1
MatrizPontos[Pallet_1,Prdt_20KitKat,1].ConfGarraOp = 0
MatrizPontos[Pallet_1,Prdt_20KitKat,1].FechaGarraOp = 0
MatrizPontos[Pallet_1,Prdt_20KitKat,1].AbreGarraOp = 0
MatrizPontos[Pallet_1,Prdt_20KitKat,1].SensoresCaixa = 123456
MatrizPontos[Pallet_1,Prdt_20KitKat,1].TravaGarra = False
MatrizPontos[Pallet_1,Prdt_20KitKat,1].SkipGoHome = False
MatrizPontos[Pallet_1,Prdt_20KitKat,1].SkipSobeRelAtual = False
MatrizPontos[Pallet_1,Prdt_20KitKat,1].XApp1Place=P1_20KitKat_1_App1
MatrizPontos[Pallet_1,Prdt_20KitKat,1].XApp2Place=P1_20KitKat_1_App2
MatrizPontos[Pallet_1,Prdt_20KitKat,1].XPlace=P1_20KitKat_1_Place
;ENDFOLD
;FOLD OffsetPlace
MatrizPontos[Pallet_1,Prdt_20KitKat,1].OffsetPlace.X=0
MatrizPontos[Pallet_1,Prdt_20KitKat,1].OffsetPlace.Y=0
MatrizPontos[Pallet_1,Prdt_20KitKat,1].OffsetPlace.Z=0
MatrizPontos[Pallet_1,Prdt_20KitKat,1].OffsetPlace.A=0
MatrizPontos[Pallet_1,Prdt_20KitKat,1].OffsetPlace.B=0
MatrizPontos[Pallet_1,Prdt_20KitKat,1].OffsetPlace.C=0
;ENDFOLD
;ENDFOLD

;FOLD PLACE 2
;FOLD PROPRIEDADES
MatrizPontos[Pallet_1,Prdt_20KitKat,2].NumCaixas = 4
MatrizPontos[Pallet_1,Prdt_20KitKat,2].PickOp = 1
MatrizPontos[Pallet_1,Prdt_20KitKat,2].ConfGarraOp = 0
MatrizPontos[Pallet_1,Prdt_20KitKat,2].FechaGarraOp = 0
MatrizPontos[Pallet_1,Prdt_20KitKat,2].AbreGarraOp = 0
MatrizPontos[Pallet_1,Prdt_20KitKat,2].SensoresCaixa = 123456
MatrizPontos[Pallet_1,Prdt_20KitKat,2].TravaGarra = False
MatrizPontos[Pallet_1,Prdt_20KitKat,2].SkipGoHome = False
MatrizPontos[Pallet_1,Prdt_20KitKat,2].SkipSobeRelAtual = False
MatrizPontos[Pallet_1,Prdt_20KitKat,2].XApp1Place=P1_20KitKat_2_App1
MatrizPontos[Pallet_1,Prdt_20KitKat,2].XApp2Place=P1_20KitKat_2_App2
MatrizPontos[Pallet_1,Prdt_20KitKat,2].XPlace=P1_20KitKat_2_Place
;ENDFOLD
;FOLD OffsetPlace
MatrizPontos[Pallet_1,Prdt_20KitKat,2].OffsetPlace.X=0
MatrizPontos[Pallet_1,Prdt_20KitKat,2].OffsetPlace.Y=0
MatrizPontos[Pallet_1,Prdt_20KitKat,2].OffsetPlace.Z=0
MatrizPontos[Pallet_1,Prdt_20KitKat,2].OffsetPlace.A=0
MatrizPontos[Pallet_1,Prdt_20KitKat,2].OffsetPlace.B=0
MatrizPontos[Pallet_1,Prdt_20KitKat,2].OffsetPlace.C=0
;ENDFOLD
;ENDFOLD

;FOLD PLACE 3
;FOLD PROPRIEDADES
MatrizPontos[Pallet_1,Prdt_20KitKat,3].NumCaixas = 4
MatrizPontos[Pallet_1,Prdt_20KitKat,3].PickOp = 1
MatrizPontos[Pallet_1,Prdt_20KitKat,3].ConfGarraOp = 0
MatrizPontos[Pallet_1,Prdt_20KitKat,3].FechaGarraOp = 0
MatrizPontos[Pallet_1,Prdt_20KitKat,3].AbreGarraOp = 0
MatrizPontos[Pallet_1,Prdt_20KitKat,3].SensoresCaixa = 123456
MatrizPontos[Pallet_1,Prdt_20KitKat,3].TravaGarra = False
MatrizPontos[Pallet_1,Prdt_20KitKat,3].SkipGoHome = False
MatrizPontos[Pallet_1,Prdt_20KitKat,3].SkipSobeRelAtual = False
MatrizPontos[Pallet_1,Prdt_20KitKat,3].XApp1Place=P1_20KitKat_3_App1
MatrizPontos[Pallet_1,Prdt_20KitKat,3].XApp2Place=P1_20KitKat_3_App2
MatrizPontos[Pallet_1,Prdt_20KitKat,3].XPlace=P1_20KitKat_3_Place
;ENDFOLD
;FOLD OffsetPlace
MatrizPontos[Pallet_1,Prdt_20KitKat,3].OffsetPlace.X=0
MatrizPontos[Pallet_1,Prdt_20KitKat,3].OffsetPlace.Y=0
MatrizPontos[Pallet_1,Prdt_20KitKat,3].OffsetPlace.Z=0
MatrizPontos[Pallet_1,Prdt_20KitKat,3].OffsetPlace.A=0
MatrizPontos[Pallet_1,Prdt_20KitKat,3].OffsetPlace.B=0
MatrizPontos[Pallet_1,Prdt_20KitKat,3].OffsetPlace.C=0
;ENDFOLD
;ENDFOLD

;ENDFOLD
;ENDFOLD

;FOLD Pallet 1 - Produto 21KitKat
;FOLD LAYER 1: PLACE 1 ate 3
;FOLD PLACE 1
;FOLD PROPRIEDADES
MatrizPontos[Pallet_1,Prdt_21KitKat,1].NumCaixas = 4
MatrizPontos[Pallet_1,Prdt_21KitKat,1].PickOp = 1
MatrizPontos[Pallet_1,Prdt_21KitKat,1].ConfGarraOp = 0
MatrizPontos[Pallet_1,Prdt_21KitKat,1].FechaGarraOp = 0
MatrizPontos[Pallet_1,Prdt_21KitKat,1].AbreGarraOp = 0
MatrizPontos[Pallet_1,Prdt_21KitKat,1].SensoresCaixa = 12345
MatrizPontos[Pallet_1,Prdt_21KitKat,1].TravaGarra = False
MatrizPontos[Pallet_1,Prdt_21KitKat,1].SkipGoHome = False
MatrizPontos[Pallet_1,Prdt_21KitKat,1].SkipSobeRelAtual = False
MatrizPontos[Pallet_1,Prdt_21KitKat,1].XApp1Place=P1_21KitKat_1_App1
MatrizPontos[Pallet_1,Prdt_21KitKat,1].XApp2Place=P1_21KitKat_1_App2
MatrizPontos[Pallet_1,Prdt_21KitKat,1].XPlace=P1_21KitKat_1_Place
;ENDFOLD
;FOLD OffsetPlace
MatrizPontos[Pallet_1,Prdt_21KitKat,1].OffsetPlace.X=0
MatrizPontos[Pallet_1,Prdt_21KitKat,1].OffsetPlace.Y=0
MatrizPontos[Pallet_1,Prdt_21KitKat,1].OffsetPlace.Z=0
MatrizPontos[Pallet_1,Prdt_21KitKat,1].OffsetPlace.A=0
MatrizPontos[Pallet_1,Prdt_21KitKat,1].OffsetPlace.B=0
MatrizPontos[Pallet_1,Prdt_21KitKat,1].OffsetPlace.C=0
;ENDFOLD
;ENDFOLD

;FOLD PLACE 2
;FOLD PROPRIEDADES
MatrizPontos[Pallet_1,Prdt_21KitKat,2].NumCaixas = 4
MatrizPontos[Pallet_1,Prdt_21KitKat,2].PickOp = 1
MatrizPontos[Pallet_1,Prdt_21KitKat,2].ConfGarraOp = 0
MatrizPontos[Pallet_1,Prdt_21KitKat,2].FechaGarraOp = 0
MatrizPontos[Pallet_1,Prdt_21KitKat,2].AbreGarraOp = 0
MatrizPontos[Pallet_1,Prdt_21KitKat,2].SensoresCaixa = 12345
MatrizPontos[Pallet_1,Prdt_21KitKat,2].TravaGarra = False
MatrizPontos[Pallet_1,Prdt_21KitKat,2].SkipGoHome = False
MatrizPontos[Pallet_1,Prdt_21KitKat,2].SkipSobeRelAtual = False
MatrizPontos[Pallet_1,Prdt_21KitKat,2].XApp1Place=P1_21KitKat_2_App1
MatrizPontos[Pallet_1,Prdt_21KitKat,2].XApp2Place=P1_21KitKat_2_App2
MatrizPontos[Pallet_1,Prdt_21KitKat,2].XPlace=P1_21KitKat_2_Place
;ENDFOLD
;FOLD OffsetPlace
MatrizPontos[Pallet_1,Prdt_21KitKat,2].OffsetPlace.X=0
MatrizPontos[Pallet_1,Prdt_21KitKat,2].OffsetPlace.Y=0
MatrizPontos[Pallet_1,Prdt_21KitKat,2].OffsetPlace.Z=0
MatrizPontos[Pallet_1,Prdt_21KitKat,2].OffsetPlace.A=0
MatrizPontos[Pallet_1,Prdt_21KitKat,2].OffsetPlace.B=0
MatrizPontos[Pallet_1,Prdt_21KitKat,2].OffsetPlace.C=0
;ENDFOLD
;ENDFOLD

;FOLD PLACE 3
;FOLD PROPRIEDADES
MatrizPontos[Pallet_1,Prdt_21KitKat,3].NumCaixas = 4
MatrizPontos[Pallet_1,Prdt_21KitKat,3].PickOp = 1
MatrizPontos[Pallet_1,Prdt_21KitKat,3].ConfGarraOp = 0
MatrizPontos[Pallet_1,Prdt_21KitKat,3].FechaGarraOp = 0
MatrizPontos[Pallet_1,Prdt_21KitKat,3].AbreGarraOp = 0
MatrizPontos[Pallet_1,Prdt_21KitKat,3].SensoresCaixa = 12345
MatrizPontos[Pallet_1,Prdt_21KitKat,3].TravaGarra = False
MatrizPontos[Pallet_1,Prdt_21KitKat,3].SkipGoHome = False
MatrizPontos[Pallet_1,Prdt_21KitKat,3].SkipSobeRelAtual = False
MatrizPontos[Pallet_1,Prdt_21KitKat,3].XApp1Place=P1_21KitKat_3_App1
MatrizPontos[Pallet_1,Prdt_21KitKat,3].XApp2Place=P1_21KitKat_3_App2
MatrizPontos[Pallet_1,Prdt_21KitKat,3].XPlace=P1_21KitKat_3_Place
;ENDFOLD
;FOLD OffsetPlace
MatrizPontos[Pallet_1,Prdt_21KitKat,3].OffsetPlace.X=0
MatrizPontos[Pallet_1,Prdt_21KitKat,3].OffsetPlace.Y=0
MatrizPontos[Pallet_1,Prdt_21KitKat,3].OffsetPlace.Z=0
MatrizPontos[Pallet_1,Prdt_21KitKat,3].OffsetPlace.A=0
MatrizPontos[Pallet_1,Prdt_21KitKat,3].OffsetPlace.B=0
MatrizPontos[Pallet_1,Prdt_21KitKat,3].OffsetPlace.C=0
;ENDFOLD
;ENDFOLD

;ENDFOLD
;ENDFOLD

;FOLD Pallet 1 - Produto 23Smarties
;FOLD LAYER 1: PLACE 1 ate 4
;FOLD PLACE 1
;FOLD PROPRIEDADES
MatrizPontos[Pallet_1,Prdt_23Smarties,1].NumCaixas = 2
MatrizPontos[Pallet_1,Prdt_23Smarties,1].PickOp = 4
MatrizPontos[Pallet_1,Prdt_23Smarties,1].ConfGarraOp = 4
MatrizPontos[Pallet_1,Prdt_23Smarties,1].FechaGarraOp = 0
MatrizPontos[Pallet_1,Prdt_23Smarties,1].AbreGarraOp = 0
MatrizPontos[Pallet_1,Prdt_23Smarties,1].SensoresCaixa = 456
MatrizPontos[Pallet_1,Prdt_23Smarties,1].TravaGarra = False
MatrizPontos[Pallet_1,Prdt_23Smarties,1].SkipGoHome = False
MatrizPontos[Pallet_1,Prdt_23Smarties,1].SkipSobeRelAtual = False
MatrizPontos[Pallet_1,Prdt_23Smarties,1].XApp1Place=P1_23Smarties_1_App1
MatrizPontos[Pallet_1,Prdt_23Smarties,1].XApp2Place=P1_23Smarties_1_App2
MatrizPontos[Pallet_1,Prdt_23Smarties,1].XPlace=P1_23Smarties_1_Place
;ENDFOLD
;FOLD OffsetPlace
MatrizPontos[Pallet_1,Prdt_23Smarties,1].OffsetPlace.X=0
MatrizPontos[Pallet_1,Prdt_23Smarties,1].OffsetPlace.Y=0
MatrizPontos[Pallet_1,Prdt_23Smarties,1].OffsetPlace.Z=0
MatrizPontos[Pallet_1,Prdt_23Smarties,1].OffsetPlace.A=0
MatrizPontos[Pallet_1,Prdt_23Smarties,1].OffsetPlace.B=0
MatrizPontos[Pallet_1,Prdt_23Smarties,1].OffsetPlace.C=0
;ENDFOLD
;ENDFOLD

;FOLD PLACE 2
;FOLD PROPRIEDADES
MatrizPontos[Pallet_1,Prdt_23Smarties,2].NumCaixas = 3
MatrizPontos[Pallet_1,Prdt_23Smarties,2].PickOp = 4
MatrizPontos[Pallet_1,Prdt_23Smarties,2].ConfGarraOp = 4
MatrizPontos[Pallet_1,Prdt_23Smarties,2].FechaGarraOp = 0
MatrizPontos[Pallet_1,Prdt_23Smarties,2].AbreGarraOp = 0
MatrizPontos[Pallet_1,Prdt_23Smarties,2].SensoresCaixa = 3456
MatrizPontos[Pallet_1,Prdt_23Smarties,2].TravaGarra = False
MatrizPontos[Pallet_1,Prdt_23Smarties,2].SkipGoHome = False
MatrizPontos[Pallet_1,Prdt_23Smarties,2].SkipSobeRelAtual = False
MatrizPontos[Pallet_1,Prdt_23Smarties,2].XApp1Place=P1_23Smarties_2_App1
MatrizPontos[Pallet_1,Prdt_23Smarties,2].XApp2Place=P1_23Smarties_2_App2
MatrizPontos[Pallet_1,Prdt_23Smarties,2].XPlace=P1_23Smarties_2_Place
;ENDFOLD
;FOLD OffsetPlace
MatrizPontos[Pallet_1,Prdt_23Smarties,2].OffsetPlace.X=0
MatrizPontos[Pallet_1,Prdt_23Smarties,2].OffsetPlace.Y=0
MatrizPontos[Pallet_1,Prdt_23Smarties,2].OffsetPlace.Z=0
MatrizPontos[Pallet_1,Prdt_23Smarties,2].OffsetPlace.A=0
MatrizPontos[Pallet_1,Prdt_23Smarties,2].OffsetPlace.B=0
MatrizPontos[Pallet_1,Prdt_23Smarties,2].OffsetPlace.C=0
;ENDFOLD
;ENDFOLD

;FOLD PLACE 3
;FOLD PROPRIEDADES
MatrizPontos[Pallet_1,Prdt_23Smarties,3].NumCaixas = 2
MatrizPontos[Pallet_1,Prdt_23Smarties,3].PickOp = 4
MatrizPontos[Pallet_1,Prdt_23Smarties,3].ConfGarraOp = 4
MatrizPontos[Pallet_1,Prdt_23Smarties,3].FechaGarraOp = 0
MatrizPontos[Pallet_1,Prdt_23Smarties,3].AbreGarraOp = 0
MatrizPontos[Pallet_1,Prdt_23Smarties,3].SensoresCaixa = 456
MatrizPontos[Pallet_1,Prdt_23Smarties,3].TravaGarra = False
MatrizPontos[Pallet_1,Prdt_23Smarties,3].SkipGoHome = False
MatrizPontos[Pallet_1,Prdt_23Smarties,3].SkipSobeRelAtual = False
MatrizPontos[Pallet_1,Prdt_23Smarties,3].XApp1Place=P1_23Smarties_3_App1
MatrizPontos[Pallet_1,Prdt_23Smarties,3].XApp2Place=P1_23Smarties_3_App2
MatrizPontos[Pallet_1,Prdt_23Smarties,3].XPlace=P1_23Smarties_3_Place
;ENDFOLD
;FOLD OffsetPlace
MatrizPontos[Pallet_1,Prdt_23Smarties,3].OffsetPlace.X=0
MatrizPontos[Pallet_1,Prdt_23Smarties,3].OffsetPlace.Y=0
MatrizPontos[Pallet_1,Prdt_23Smarties,3].OffsetPlace.Z=0
MatrizPontos[Pallet_1,Prdt_23Smarties,3].OffsetPlace.A=0
MatrizPontos[Pallet_1,Prdt_23Smarties,3].OffsetPlace.B=0
MatrizPontos[Pallet_1,Prdt_23Smarties,3].OffsetPlace.C=0
;ENDFOLD
;ENDFOLD

;FOLD PLACE 4
;FOLD PROPRIEDADES
MatrizPontos[Pallet_1,Prdt_23Smarties,4].NumCaixas = 3
MatrizPontos[Pallet_1,Prdt_23Smarties,4].PickOp = 4
MatrizPontos[Pallet_1,Prdt_23Smarties,4].ConfGarraOp = 4
MatrizPontos[Pallet_1,Prdt_23Smarties,4].FechaGarraOp = 0
MatrizPontos[Pallet_1,Prdt_23Smarties,4].AbreGarraOp = 0
MatrizPontos[Pallet_1,Prdt_23Smarties,4].SensoresCaixa = 3456
MatrizPontos[Pallet_1,Prdt_23Smarties,4].TravaGarra = False
MatrizPontos[Pallet_1,Prdt_23Smarties,4].SkipGoHome = False
MatrizPontos[Pallet_1,Prdt_23Smarties,4].SkipSobeRelAtual = False
MatrizPontos[Pallet_1,Prdt_23Smarties,4].XApp1Place=P1_23Smarties_4_App1
MatrizPontos[Pallet_1,Prdt_23Smarties,4].XApp2Place=P1_23Smarties_4_App2
MatrizPontos[Pallet_1,Prdt_23Smarties,4].XPlace=P1_23Smarties_4_Place
;ENDFOLD
;FOLD OffsetPlace
MatrizPontos[Pallet_1,Prdt_23Smarties,4].OffsetPlace.X=0
MatrizPontos[Pallet_1,Prdt_23Smarties,4].OffsetPlace.Y=0
MatrizPontos[Pallet_1,Prdt_23Smarties,4].OffsetPlace.Z=0
MatrizPontos[Pallet_1,Prdt_23Smarties,4].OffsetPlace.A=0
MatrizPontos[Pallet_1,Prdt_23Smarties,4].OffsetPlace.B=0
MatrizPontos[Pallet_1,Prdt_23Smarties,4].OffsetPlace.C=0
;ENDFOLD
;ENDFOLD

;ENDFOLD
;FOLD LAYER 2: PLACE 5 ate 8
;FOLD PLACE 5
;FOLD PROPRIEDADES
MatrizPontos[Pallet_1,Prdt_23Smarties,5].NumCaixas = 2
MatrizPontos[Pallet_1,Prdt_23Smarties,5].PickOp = 5
MatrizPontos[Pallet_1,Prdt_23Smarties,5].ConfGarraOp = 4
MatrizPontos[Pallet_1,Prdt_23Smarties,5].FechaGarraOp = 0
MatrizPontos[Pallet_1,Prdt_23Smarties,5].AbreGarraOp = 0
MatrizPontos[Pallet_1,Prdt_23Smarties,5].SensoresCaixa = 123
MatrizPontos[Pallet_1,Prdt_23Smarties,5].TravaGarra = False
MatrizPontos[Pallet_1,Prdt_23Smarties,5].SkipGoHome = False
MatrizPontos[Pallet_1,Prdt_23Smarties,5].SkipSobeRelAtual = False
MatrizPontos[Pallet_1,Prdt_23Smarties,5].XApp1Place=P1_23Smarties_5_App1
MatrizPontos[Pallet_1,Prdt_23Smarties,5].XApp2Place=P1_23Smarties_5_App2
MatrizPontos[Pallet_1,Prdt_23Smarties,5].XPlace=P1_23Smarties_5_Place
;ENDFOLD
;FOLD OffsetPlace
MatrizPontos[Pallet_1,Prdt_23Smarties,5].OffsetPlace.X=0
MatrizPontos[Pallet_1,Prdt_23Smarties,5].OffsetPlace.Y=0
MatrizPontos[Pallet_1,Prdt_23Smarties,5].OffsetPlace.Z=0
MatrizPontos[Pallet_1,Prdt_23Smarties,5].OffsetPlace.A=0
MatrizPontos[Pallet_1,Prdt_23Smarties,5].OffsetPlace.B=0
MatrizPontos[Pallet_1,Prdt_23Smarties,5].OffsetPlace.C=0
;ENDFOLD
;ENDFOLD

;FOLD PLACE 6
;FOLD PROPRIEDADES
MatrizPontos[Pallet_1,Prdt_23Smarties,6].NumCaixas = 3
MatrizPontos[Pallet_1,Prdt_23Smarties,6].PickOp = 5
MatrizPontos[Pallet_1,Prdt_23Smarties,6].ConfGarraOp = 4
MatrizPontos[Pallet_1,Prdt_23Smarties,6].FechaGarraOp = 0
MatrizPontos[Pallet_1,Prdt_23Smarties,6].AbreGarraOp = 0
MatrizPontos[Pallet_1,Prdt_23Smarties,6].SensoresCaixa = 1234
MatrizPontos[Pallet_1,Prdt_23Smarties,6].TravaGarra = False
MatrizPontos[Pallet_1,Prdt_23Smarties,6].SkipGoHome = False
MatrizPontos[Pallet_1,Prdt_23Smarties,6].SkipSobeRelAtual = False
MatrizPontos[Pallet_1,Prdt_23Smarties,6].XApp1Place=P1_23Smarties_6_App1
MatrizPontos[Pallet_1,Prdt_23Smarties,6].XApp2Place=P1_23Smarties_6_App2
MatrizPontos[Pallet_1,Prdt_23Smarties,6].XPlace=P1_23Smarties_6_Place
;ENDFOLD
;FOLD OffsetPlace
MatrizPontos[Pallet_1,Prdt_23Smarties,6].OffsetPlace.X=0
MatrizPontos[Pallet_1,Prdt_23Smarties,6].OffsetPlace.Y=0
MatrizPontos[Pallet_1,Prdt_23Smarties,6].OffsetPlace.Z=0
MatrizPontos[Pallet_1,Prdt_23Smarties,6].OffsetPlace.A=0
MatrizPontos[Pallet_1,Prdt_23Smarties,6].OffsetPlace.B=0
MatrizPontos[Pallet_1,Prdt_23Smarties,6].OffsetPlace.C=0
;ENDFOLD
;ENDFOLD

;FOLD PLACE 7
;FOLD PROPRIEDADES
MatrizPontos[Pallet_1,Prdt_23Smarties,7].NumCaixas = 2
MatrizPontos[Pallet_1,Prdt_23Smarties,7].PickOp = 5
MatrizPontos[Pallet_1,Prdt_23Smarties,7].ConfGarraOp = 4
MatrizPontos[Pallet_1,Prdt_23Smarties,7].FechaGarraOp = 0
MatrizPontos[Pallet_1,Prdt_23Smarties,7].AbreGarraOp = 0
MatrizPontos[Pallet_1,Prdt_23Smarties,7].SensoresCaixa = 123
MatrizPontos[Pallet_1,Prdt_23Smarties,7].TravaGarra = False
MatrizPontos[Pallet_1,Prdt_23Smarties,7].SkipGoHome = False
MatrizPontos[Pallet_1,Prdt_23Smarties,7].SkipSobeRelAtual = False
MatrizPontos[Pallet_1,Prdt_23Smarties,7].XApp1Place=P1_23Smarties_7_App1
MatrizPontos[Pallet_1,Prdt_23Smarties,7].XApp2Place=P1_23Smarties_7_App2
MatrizPontos[Pallet_1,Prdt_23Smarties,7].XPlace=P1_23Smarties_7_Place
;ENDFOLD
;FOLD OffsetPlace
MatrizPontos[Pallet_1,Prdt_23Smarties,7].OffsetPlace.X=0
MatrizPontos[Pallet_1,Prdt_23Smarties,7].OffsetPlace.Y=0
MatrizPontos[Pallet_1,Prdt_23Smarties,7].OffsetPlace.Z=0
MatrizPontos[Pallet_1,Prdt_23Smarties,7].OffsetPlace.A=0
MatrizPontos[Pallet_1,Prdt_23Smarties,7].OffsetPlace.B=0
MatrizPontos[Pallet_1,Prdt_23Smarties,7].OffsetPlace.C=0
;ENDFOLD
;ENDFOLD

;FOLD PLACE 8
;FOLD PROPRIEDADES
MatrizPontos[Pallet_1,Prdt_23Smarties,8].NumCaixas = 3
MatrizPontos[Pallet_1,Prdt_23Smarties,8].PickOp = 5
MatrizPontos[Pallet_1,Prdt_23Smarties,8].ConfGarraOp = 4
MatrizPontos[Pallet_1,Prdt_23Smarties,8].FechaGarraOp = 0
MatrizPontos[Pallet_1,Prdt_23Smarties,8].AbreGarraOp = 0
MatrizPontos[Pallet_1,Prdt_23Smarties,8].SensoresCaixa = 1234
MatrizPontos[Pallet_1,Prdt_23Smarties,8].TravaGarra = False
MatrizPontos[Pallet_1,Prdt_23Smarties,8].SkipGoHome = False
MatrizPontos[Pallet_1,Prdt_23Smarties,8].SkipSobeRelAtual = False
MatrizPontos[Pallet_1,Prdt_23Smarties,8].XApp1Place=P1_23Smarties_8_App1
MatrizPontos[Pallet_1,Prdt_23Smarties,8].XApp2Place=P1_23Smarties_8_App2
MatrizPontos[Pallet_1,Prdt_23Smarties,8].XPlace=P1_23Smarties_8_Place
;ENDFOLD
;FOLD OffsetPlace
MatrizPontos[Pallet_1,Prdt_23Smarties,8].OffsetPlace.X=0
MatrizPontos[Pallet_1,Prdt_23Smarties,8].OffsetPlace.Y=0
MatrizPontos[Pallet_1,Prdt_23Smarties,8].OffsetPlace.Z=0
MatrizPontos[Pallet_1,Prdt_23Smarties,8].OffsetPlace.A=0
MatrizPontos[Pallet_1,Prdt_23Smarties,8].OffsetPlace.B=0
MatrizPontos[Pallet_1,Prdt_23Smarties,8].OffsetPlace.C=0
;ENDFOLD
;ENDFOLD

;ENDFOLD
;ENDFOLD

;FOLD Pallet 1 - Produto 22KitKat
;FOLD LAYER 1: PLACE 1 ate 4
;FOLD PLACE 1
;FOLD PROPRIEDADES
MatrizPontos[Pallet_1,Prdt_22KitKat,1].NumCaixas = 2
MatrizPontos[Pallet_1,Prdt_22KitKat,1].PickOp = 2
MatrizPontos[Pallet_1,Prdt_22KitKat,1].ConfGarraOp = 2
MatrizPontos[Pallet_1,Prdt_22KitKat,1].FechaGarraOp = 0
MatrizPontos[Pallet_1,Prdt_22KitKat,1].AbreGarraOp = 0
MatrizPontos[Pallet_1,Prdt_22KitKat,1].SensoresCaixa = 123
MatrizPontos[Pallet_1,Prdt_22KitKat,1].TravaGarra = False
MatrizPontos[Pallet_1,Prdt_22KitKat,1].SkipGoHome = False
MatrizPontos[Pallet_1,Prdt_22KitKat,1].SkipSobeRelAtual = False
MatrizPontos[Pallet_1,Prdt_22KitKat,1].XApp1Place=P1_22KitKat_1_App1
MatrizPontos[Pallet_1,Prdt_22KitKat,1].XApp2Place=P1_22KitKat_1_App2
MatrizPontos[Pallet_1,Prdt_22KitKat,1].XPlace=P1_22KitKat_1_Place
;ENDFOLD
;FOLD OffsetPlace
MatrizPontos[Pallet_1,Prdt_22KitKat,1].OffsetPlace.X=0
MatrizPontos[Pallet_1,Prdt_22KitKat,1].OffsetPlace.Y=0
MatrizPontos[Pallet_1,Prdt_22KitKat,1].OffsetPlace.Z=0
MatrizPontos[Pallet_1,Prdt_22KitKat,1].OffsetPlace.A=0
MatrizPontos[Pallet_1,Prdt_22KitKat,1].OffsetPlace.B=0
MatrizPontos[Pallet_1,Prdt_22KitKat,1].OffsetPlace.C=0
;ENDFOLD
;ENDFOLD

;FOLD PLACE 2
;FOLD PROPRIEDADES
MatrizPontos[Pallet_1,Prdt_22KitKat,2].NumCaixas = 2
MatrizPontos[Pallet_1,Prdt_22KitKat,2].PickOp = 2
MatrizPontos[Pallet_1,Prdt_22KitKat,2].ConfGarraOp = 2
MatrizPontos[Pallet_1,Prdt_22KitKat,2].FechaGarraOp = 0
MatrizPontos[Pallet_1,Prdt_22KitKat,2].AbreGarraOp = 0
MatrizPontos[Pallet_1,Prdt_22KitKat,2].SensoresCaixa = 123
MatrizPontos[Pallet_1,Prdt_22KitKat,2].TravaGarra = False
MatrizPontos[Pallet_1,Prdt_22KitKat,2].SkipGoHome = False
MatrizPontos[Pallet_1,Prdt_22KitKat,2].SkipSobeRelAtual = False
MatrizPontos[Pallet_1,Prdt_22KitKat,2].XApp1Place=P1_22KitKat_2_App1
MatrizPontos[Pallet_1,Prdt_22KitKat,2].XApp2Place=P1_22KitKat_2_App2
MatrizPontos[Pallet_1,Prdt_22KitKat,2].XPlace=P1_22KitKat_2_Place
;ENDFOLD
;FOLD OffsetPlace
MatrizPontos[Pallet_1,Prdt_22KitKat,2].OffsetPlace.X=0
MatrizPontos[Pallet_1,Prdt_22KitKat,2].OffsetPlace.Y=0
MatrizPontos[Pallet_1,Prdt_22KitKat,2].OffsetPlace.Z=0
MatrizPontos[Pallet_1,Prdt_22KitKat,2].OffsetPlace.A=0
MatrizPontos[Pallet_1,Prdt_22KitKat,2].OffsetPlace.B=0
MatrizPontos[Pallet_1,Prdt_22KitKat,2].OffsetPlace.C=0
;ENDFOLD
;ENDFOLD

;FOLD PLACE 3
;FOLD PROPRIEDADES
MatrizPontos[Pallet_1,Prdt_22KitKat,3].NumCaixas = 2
MatrizPontos[Pallet_1,Prdt_22KitKat,3].PickOp = 2
MatrizPontos[Pallet_1,Prdt_22KitKat,3].ConfGarraOp = 2
MatrizPontos[Pallet_1,Prdt_22KitKat,3].FechaGarraOp = 0
MatrizPontos[Pallet_1,Prdt_22KitKat,3].AbreGarraOp = 0
MatrizPontos[Pallet_1,Prdt_22KitKat,3].SensoresCaixa = 123
MatrizPontos[Pallet_1,Prdt_22KitKat,3].TravaGarra = False
MatrizPontos[Pallet_1,Prdt_22KitKat,3].SkipGoHome = False
MatrizPontos[Pallet_1,Prdt_22KitKat,3].SkipSobeRelAtual = False
MatrizPontos[Pallet_1,Prdt_22KitKat,3].XApp1Place=P1_22KitKat_3_App1
MatrizPontos[Pallet_1,Prdt_22KitKat,3].XApp2Place=P1_22KitKat_3_App2
MatrizPontos[Pallet_1,Prdt_22KitKat,3].XPlace=P1_22KitKat_3_Place
;ENDFOLD
;FOLD OffsetPlace
MatrizPontos[Pallet_1,Prdt_22KitKat,3].OffsetPlace.X=0
MatrizPontos[Pallet_1,Prdt_22KitKat,3].OffsetPlace.Y=0
MatrizPontos[Pallet_1,Prdt_22KitKat,3].OffsetPlace.Z=0
MatrizPontos[Pallet_1,Prdt_22KitKat,3].OffsetPlace.A=0
MatrizPontos[Pallet_1,Prdt_22KitKat,3].OffsetPlace.B=0
MatrizPontos[Pallet_1,Prdt_22KitKat,3].OffsetPlace.C=0
;ENDFOLD
;ENDFOLD

;FOLD PLACE 4
;FOLD PROPRIEDADES
MatrizPontos[Pallet_1,Prdt_22KitKat,4].NumCaixas = 4
MatrizPontos[Pallet_1,Prdt_22KitKat,4].PickOp = 2
MatrizPontos[Pallet_1,Prdt_22KitKat,4].ConfGarraOp = 2
MatrizPontos[Pallet_1,Prdt_22KitKat,4].FechaGarraOp = 0
MatrizPontos[Pallet_1,Prdt_22KitKat,4].AbreGarraOp = 0
MatrizPontos[Pallet_1,Prdt_22KitKat,4].SensoresCaixa = 123456
MatrizPontos[Pallet_1,Prdt_22KitKat,4].TravaGarra = False
MatrizPontos[Pallet_1,Prdt_22KitKat,4].SkipGoHome = False
MatrizPontos[Pallet_1,Prdt_22KitKat,4].SkipSobeRelAtual = False
MatrizPontos[Pallet_1,Prdt_22KitKat,4].XApp1Place=P1_22KitKat_4_App1
MatrizPontos[Pallet_1,Prdt_22KitKat,4].XApp2Place=P1_22KitKat_4_App2
MatrizPontos[Pallet_1,Prdt_22KitKat,4].XPlace=P1_22KitKat_4_Place
;ENDFOLD
;FOLD OffsetPlace
MatrizPontos[Pallet_1,Prdt_22KitKat,4].OffsetPlace.X=0
MatrizPontos[Pallet_1,Prdt_22KitKat,4].OffsetPlace.Y=0
MatrizPontos[Pallet_1,Prdt_22KitKat,4].OffsetPlace.Z=0
MatrizPontos[Pallet_1,Prdt_22KitKat,4].OffsetPlace.A=0
MatrizPontos[Pallet_1,Prdt_22KitKat,4].OffsetPlace.B=0
MatrizPontos[Pallet_1,Prdt_22KitKat,4].OffsetPlace.C=0
;ENDFOLD
;ENDFOLD

;ENDFOLD
;FOLD LAYER 2: PLACE 5 ate 8
;FOLD PLACE 5
;FOLD PROPRIEDADES
MatrizPontos[Pallet_1,Prdt_22KitKat,5].NumCaixas = 4
MatrizPontos[Pallet_1,Prdt_22KitKat,5].PickOp = 2
MatrizPontos[Pallet_1,Prdt_22KitKat,5].ConfGarraOp = 2
MatrizPontos[Pallet_1,Prdt_22KitKat,5].FechaGarraOp = 0
MatrizPontos[Pallet_1,Prdt_22KitKat,5].AbreGarraOp = 0
MatrizPontos[Pallet_1,Prdt_22KitKat,5].SensoresCaixa = 123456
MatrizPontos[Pallet_1,Prdt_22KitKat,5].TravaGarra = False
MatrizPontos[Pallet_1,Prdt_22KitKat,5].SkipGoHome = False
MatrizPontos[Pallet_1,Prdt_22KitKat,5].SkipSobeRelAtual = False
MatrizPontos[Pallet_1,Prdt_22KitKat,5].XApp1Place=P1_22KitKat_5_App1
MatrizPontos[Pallet_1,Prdt_22KitKat,5].XApp2Place=P1_22KitKat_5_App2
MatrizPontos[Pallet_1,Prdt_22KitKat,5].XPlace=P1_22KitKat_5_Place
;ENDFOLD
;FOLD OffsetPlace
MatrizPontos[Pallet_1,Prdt_22KitKat,5].OffsetPlace.X=0
MatrizPontos[Pallet_1,Prdt_22KitKat,5].OffsetPlace.Y=0
MatrizPontos[Pallet_1,Prdt_22KitKat,5].OffsetPlace.Z=0
MatrizPontos[Pallet_1,Prdt_22KitKat,5].OffsetPlace.A=0
MatrizPontos[Pallet_1,Prdt_22KitKat,5].OffsetPlace.B=0
MatrizPontos[Pallet_1,Prdt_22KitKat,5].OffsetPlace.C=0
;ENDFOLD
;ENDFOLD

;FOLD PLACE 6
;FOLD PROPRIEDADES
MatrizPontos[Pallet_1,Prdt_22KitKat,6].NumCaixas = 2
MatrizPontos[Pallet_1,Prdt_22KitKat,6].PickOp = 2
MatrizPontos[Pallet_1,Prdt_22KitKat,6].ConfGarraOp = 2
MatrizPontos[Pallet_1,Prdt_22KitKat,6].FechaGarraOp = 0
MatrizPontos[Pallet_1,Prdt_22KitKat,6].AbreGarraOp = 0
MatrizPontos[Pallet_1,Prdt_22KitKat,6].SensoresCaixa = 123
MatrizPontos[Pallet_1,Prdt_22KitKat,6].TravaGarra = False
MatrizPontos[Pallet_1,Prdt_22KitKat,6].SkipGoHome = False
MatrizPontos[Pallet_1,Prdt_22KitKat,6].SkipSobeRelAtual = False
MatrizPontos[Pallet_1,Prdt_22KitKat,6].XApp1Place=P1_22KitKat_6_App1
MatrizPontos[Pallet_1,Prdt_22KitKat,6].XApp2Place=P1_22KitKat_6_App2
MatrizPontos[Pallet_1,Prdt_22KitKat,6].XPlace=P1_22KitKat_6_Place
;ENDFOLD
;FOLD OffsetPlace
MatrizPontos[Pallet_1,Prdt_22KitKat,6].OffsetPlace.X=0
MatrizPontos[Pallet_1,Prdt_22KitKat,6].OffsetPlace.Y=0
MatrizPontos[Pallet_1,Prdt_22KitKat,6].OffsetPlace.Z=0
MatrizPontos[Pallet_1,Prdt_22KitKat,6].OffsetPlace.A=0
MatrizPontos[Pallet_1,Prdt_22KitKat,6].OffsetPlace.B=0
MatrizPontos[Pallet_1,Prdt_22KitKat,6].OffsetPlace.C=0
;ENDFOLD
;ENDFOLD

;FOLD PLACE 7
;FOLD PROPRIEDADES
MatrizPontos[Pallet_1,Prdt_22KitKat,7].NumCaixas = 2
MatrizPontos[Pallet_1,Prdt_22KitKat,7].PickOp = 2
MatrizPontos[Pallet_1,Prdt_22KitKat,7].ConfGarraOp = 2
MatrizPontos[Pallet_1,Prdt_22KitKat,7].FechaGarraOp = 0
MatrizPontos[Pallet_1,Prdt_22KitKat,7].AbreGarraOp = 0
MatrizPontos[Pallet_1,Prdt_22KitKat,7].SensoresCaixa = 123
MatrizPontos[Pallet_1,Prdt_22KitKat,7].TravaGarra = False
MatrizPontos[Pallet_1,Prdt_22KitKat,7].SkipGoHome = False
MatrizPontos[Pallet_1,Prdt_22KitKat,7].SkipSobeRelAtual = False
MatrizPontos[Pallet_1,Prdt_22KitKat,7].XApp1Place=P1_22KitKat_7_App1
MatrizPontos[Pallet_1,Prdt_22KitKat,7].XApp2Place=P1_22KitKat_7_App2
MatrizPontos[Pallet_1,Prdt_22KitKat,7].XPlace=P1_22KitKat_7_Place
;ENDFOLD
;FOLD OffsetPlace
MatrizPontos[Pallet_1,Prdt_22KitKat,7].OffsetPlace.X=0
MatrizPontos[Pallet_1,Prdt_22KitKat,7].OffsetPlace.Y=0
MatrizPontos[Pallet_1,Prdt_22KitKat,7].OffsetPlace.Z=0
MatrizPontos[Pallet_1,Prdt_22KitKat,7].OffsetPlace.A=0
MatrizPontos[Pallet_1,Prdt_22KitKat,7].OffsetPlace.B=0
MatrizPontos[Pallet_1,Prdt_22KitKat,7].OffsetPlace.C=0
;ENDFOLD
;ENDFOLD

;FOLD PLACE 8
;FOLD PROPRIEDADES
MatrizPontos[Pallet_1,Prdt_22KitKat,8].NumCaixas = 2
MatrizPontos[Pallet_1,Prdt_22KitKat,8].PickOp = 2
MatrizPontos[Pallet_1,Prdt_22KitKat,8].ConfGarraOp = 2
MatrizPontos[Pallet_1,Prdt_22KitKat,8].FechaGarraOp = 0
MatrizPontos[Pallet_1,Prdt_22KitKat,8].AbreGarraOp = 0
MatrizPontos[Pallet_1,Prdt_22KitKat,8].SensoresCaixa = 123
MatrizPontos[Pallet_1,Prdt_22KitKat,8].TravaGarra = False
MatrizPontos[Pallet_1,Prdt_22KitKat,8].SkipGoHome = False
MatrizPontos[Pallet_1,Prdt_22KitKat,8].SkipSobeRelAtual = False
MatrizPontos[Pallet_1,Prdt_22KitKat,8].XApp1Place=P1_22KitKat_8_App1
MatrizPontos[Pallet_1,Prdt_22KitKat,8].XApp2Place=P1_22KitKat_8_App2
MatrizPontos[Pallet_1,Prdt_22KitKat,8].XPlace=P1_22KitKat_8_Place
;ENDFOLD
;FOLD OffsetPlace
MatrizPontos[Pallet_1,Prdt_22KitKat,8].OffsetPlace.X=0
MatrizPontos[Pallet_1,Prdt_22KitKat,8].OffsetPlace.Y=0
MatrizPontos[Pallet_1,Prdt_22KitKat,8].OffsetPlace.Z=0
MatrizPontos[Pallet_1,Prdt_22KitKat,8].OffsetPlace.A=0
MatrizPontos[Pallet_1,Prdt_22KitKat,8].OffsetPlace.B=0
MatrizPontos[Pallet_1,Prdt_22KitKat,8].OffsetPlace.C=0
;ENDFOLD
;ENDFOLD

;ENDFOLD
;ENDFOLD

;FOLD Pallet 1 - Produto 24a28All
;FOLD LAYER 1: PLACE 1 ate 3
;FOLD PLACE 1
;FOLD PROPRIEDADES
MatrizPontos[Pallet_1,Prdt_24a28All,1].NumCaixas = 5
MatrizPontos[Pallet_1,Prdt_24a28All,1].PickOp = 1
MatrizPontos[Pallet_1,Prdt_24a28All,1].ConfGarraOp = 0
MatrizPontos[Pallet_1,Prdt_24a28All,1].FechaGarraOp = 0
MatrizPontos[Pallet_1,Prdt_24a28All,1].AbreGarraOp = 0
MatrizPontos[Pallet_1,Prdt_24a28All,1].SensoresCaixa = 123456
MatrizPontos[Pallet_1,Prdt_24a28All,1].TravaGarra = False
MatrizPontos[Pallet_1,Prdt_24a28All,1].SkipGoHome = False
MatrizPontos[Pallet_1,Prdt_24a28All,1].SkipSobeRelAtual = False
MatrizPontos[Pallet_1,Prdt_24a28All,1].XApp1Place=P1_24a28All_1_App1
MatrizPontos[Pallet_1,Prdt_24a28All,1].XApp2Place=P1_24a28All_1_App2
MatrizPontos[Pallet_1,Prdt_24a28All,1].XPlace=P1_24a28All_1_Place
;ENDFOLD
;FOLD OffsetPlace
MatrizPontos[Pallet_1,Prdt_24a28All,1].OffsetPlace.X=0
MatrizPontos[Pallet_1,Prdt_24a28All,1].OffsetPlace.Y=0
MatrizPontos[Pallet_1,Prdt_24a28All,1].OffsetPlace.Z=0
MatrizPontos[Pallet_1,Prdt_24a28All,1].OffsetPlace.A=0
MatrizPontos[Pallet_1,Prdt_24a28All,1].OffsetPlace.B=0
MatrizPontos[Pallet_1,Prdt_24a28All,1].OffsetPlace.C=0
;ENDFOLD
;ENDFOLD

;FOLD PLACE 2
;FOLD PROPRIEDADES
MatrizPontos[Pallet_1,Prdt_24a28All,2].NumCaixas = 5
MatrizPontos[Pallet_1,Prdt_24a28All,2].PickOp = 1
MatrizPontos[Pallet_1,Prdt_24a28All,2].ConfGarraOp = 0
MatrizPontos[Pallet_1,Prdt_24a28All,2].FechaGarraOp = 0
MatrizPontos[Pallet_1,Prdt_24a28All,2].AbreGarraOp = 0
MatrizPontos[Pallet_1,Prdt_24a28All,2].SensoresCaixa = 123456
MatrizPontos[Pallet_1,Prdt_24a28All,2].TravaGarra = False
MatrizPontos[Pallet_1,Prdt_24a28All,2].SkipGoHome = False
MatrizPontos[Pallet_1,Prdt_24a28All,2].SkipSobeRelAtual = False
MatrizPontos[Pallet_1,Prdt_24a28All,2].XApp1Place=P1_24a28All_2_App1
MatrizPontos[Pallet_1,Prdt_24a28All,2].XApp2Place=P1_24a28All_2_App2
MatrizPontos[Pallet_1,Prdt_24a28All,2].XPlace=P1_24a28All_2_Place
;ENDFOLD
;FOLD OffsetPlace
MatrizPontos[Pallet_1,Prdt_24a28All,2].OffsetPlace.X=0
MatrizPontos[Pallet_1,Prdt_24a28All,2].OffsetPlace.Y=0
MatrizPontos[Pallet_1,Prdt_24a28All,2].OffsetPlace.Z=0
MatrizPontos[Pallet_1,Prdt_24a28All,2].OffsetPlace.A=0
MatrizPontos[Pallet_1,Prdt_24a28All,2].OffsetPlace.B=0
MatrizPontos[Pallet_1,Prdt_24a28All,2].OffsetPlace.C=0
;ENDFOLD
;ENDFOLD

;FOLD PLACE 3
;FOLD PROPRIEDADES
MatrizPontos[Pallet_1,Prdt_24a28All,3].NumCaixas = 5
MatrizPontos[Pallet_1,Prdt_24a28All,3].PickOp = 1
MatrizPontos[Pallet_1,Prdt_24a28All,3].ConfGarraOp = 0
MatrizPontos[Pallet_1,Prdt_24a28All,3].FechaGarraOp = 0
MatrizPontos[Pallet_1,Prdt_24a28All,3].AbreGarraOp = 0
MatrizPontos[Pallet_1,Prdt_24a28All,3].SensoresCaixa = 123456
MatrizPontos[Pallet_1,Prdt_24a28All,3].TravaGarra = False
MatrizPontos[Pallet_1,Prdt_24a28All,3].SkipGoHome = False
MatrizPontos[Pallet_1,Prdt_24a28All,3].SkipSobeRelAtual = False
MatrizPontos[Pallet_1,Prdt_24a28All,3].XApp1Place=P1_24a28All_3_App1
MatrizPontos[Pallet_1,Prdt_24a28All,3].XApp2Place=P1_24a28All_3_App2
MatrizPontos[Pallet_1,Prdt_24a28All,3].XPlace=P1_24a28All_3_Place
;ENDFOLD
;FOLD OffsetPlace
MatrizPontos[Pallet_1,Prdt_24a28All,3].OffsetPlace.X=0
MatrizPontos[Pallet_1,Prdt_24a28All,3].OffsetPlace.Y=0
MatrizPontos[Pallet_1,Prdt_24a28All,3].OffsetPlace.Z=0
MatrizPontos[Pallet_1,Prdt_24a28All,3].OffsetPlace.A=0
MatrizPontos[Pallet_1,Prdt_24a28All,3].OffsetPlace.B=0
MatrizPontos[Pallet_1,Prdt_24a28All,3].OffsetPlace.C=0
;ENDFOLD
;ENDFOLD

;ENDFOLD
;ENDFOLD

;FOLD Pallet 1 - Produto 30All
;FOLD LAYER 1: PLACE 1 ate 4
;FOLD PLACE 1
;FOLD PROPRIEDADES
MatrizPontos[Pallet_1,Prdt_30All,1].NumCaixas = 4
MatrizPontos[Pallet_1,Prdt_30All,1].PickOp = 1
MatrizPontos[Pallet_1,Prdt_30All,1].ConfGarraOp = 0
MatrizPontos[Pallet_1,Prdt_30All,1].FechaGarraOp = 0
MatrizPontos[Pallet_1,Prdt_30All,1].AbreGarraOp = 0
MatrizPontos[Pallet_1,Prdt_30All,1].SensoresCaixa = 12345
MatrizPontos[Pallet_1,Prdt_30All,1].TravaGarra = False
MatrizPontos[Pallet_1,Prdt_30All,1].SkipGoHome = False
MatrizPontos[Pallet_1,Prdt_30All,1].SkipSobeRelAtual = False
MatrizPontos[Pallet_1,Prdt_30All,1].XApp1Place=P1_30All_1_App1
MatrizPontos[Pallet_1,Prdt_30All,1].XApp2Place=P1_30All_1_App2
MatrizPontos[Pallet_1,Prdt_30All,1].XPlace=P1_30All_1_Place
;ENDFOLD
;FOLD OffsetPlace
MatrizPontos[Pallet_1,Prdt_30All,1].OffsetPlace.X=0
MatrizPontos[Pallet_1,Prdt_30All,1].OffsetPlace.Y=0
MatrizPontos[Pallet_1,Prdt_30All,1].OffsetPlace.Z=0
MatrizPontos[Pallet_1,Prdt_30All,1].OffsetPlace.A=0
MatrizPontos[Pallet_1,Prdt_30All,1].OffsetPlace.B=0
MatrizPontos[Pallet_1,Prdt_30All,1].OffsetPlace.C=0
;ENDFOLD
;ENDFOLD

;FOLD PLACE 2
;FOLD PROPRIEDADES
MatrizPontos[Pallet_1,Prdt_30All,2].NumCaixas = 4
MatrizPontos[Pallet_1,Prdt_30All,2].PickOp = 1
MatrizPontos[Pallet_1,Prdt_30All,2].ConfGarraOp = 0
MatrizPontos[Pallet_1,Prdt_30All,2].FechaGarraOp = 0
MatrizPontos[Pallet_1,Prdt_30All,2].AbreGarraOp = 0
MatrizPontos[Pallet_1,Prdt_30All,2].SensoresCaixa = 12345
MatrizPontos[Pallet_1,Prdt_30All,2].TravaGarra = False
MatrizPontos[Pallet_1,Prdt_30All,2].SkipGoHome = False
MatrizPontos[Pallet_1,Prdt_30All,2].SkipSobeRelAtual = False
MatrizPontos[Pallet_1,Prdt_30All,2].XApp1Place=P1_30All_2_App1
MatrizPontos[Pallet_1,Prdt_30All,2].XApp2Place=P1_30All_2_App2
MatrizPontos[Pallet_1,Prdt_30All,2].XPlace=P1_30All_2_Place
;ENDFOLD
;FOLD OffsetPlace
MatrizPontos[Pallet_1,Prdt_30All,2].OffsetPlace.X=0
MatrizPontos[Pallet_1,Prdt_30All,2].OffsetPlace.Y=0
MatrizPontos[Pallet_1,Prdt_30All,2].OffsetPlace.Z=0
MatrizPontos[Pallet_1,Prdt_30All,2].OffsetPlace.A=0
MatrizPontos[Pallet_1,Prdt_30All,2].OffsetPlace.B=0
MatrizPontos[Pallet_1,Prdt_30All,2].OffsetPlace.C=0
;ENDFOLD
;ENDFOLD

;FOLD PLACE 3
;FOLD PROPRIEDADES
MatrizPontos[Pallet_1,Prdt_30All,3].NumCaixas = 4
MatrizPontos[Pallet_1,Prdt_30All,3].PickOp = 1
MatrizPontos[Pallet_1,Prdt_30All,3].ConfGarraOp = 0
MatrizPontos[Pallet_1,Prdt_30All,3].FechaGarraOp = 0
MatrizPontos[Pallet_1,Prdt_30All,3].AbreGarraOp = 0
MatrizPontos[Pallet_1,Prdt_30All,3].SensoresCaixa = 12345
MatrizPontos[Pallet_1,Prdt_30All,3].TravaGarra = False
MatrizPontos[Pallet_1,Prdt_30All,3].SkipGoHome = False
MatrizPontos[Pallet_1,Prdt_30All,3].SkipSobeRelAtual = False
MatrizPontos[Pallet_1,Prdt_30All,3].XApp1Place=P1_30All_3_App1
MatrizPontos[Pallet_1,Prdt_30All,3].XApp2Place=P1_30All_3_App2
MatrizPontos[Pallet_1,Prdt_30All,3].XPlace=P1_30All_3_Place
;ENDFOLD
;FOLD OffsetPlace
MatrizPontos[Pallet_1,Prdt_30All,3].OffsetPlace.X=0
MatrizPontos[Pallet_1,Prdt_30All,3].OffsetPlace.Y=0
MatrizPontos[Pallet_1,Prdt_30All,3].OffsetPlace.Z=0
MatrizPontos[Pallet_1,Prdt_30All,3].OffsetPlace.A=0
MatrizPontos[Pallet_1,Prdt_30All,3].OffsetPlace.B=0
MatrizPontos[Pallet_1,Prdt_30All,3].OffsetPlace.C=0
;ENDFOLD
;ENDFOLD

;FOLD PLACE 4
;FOLD PROPRIEDADES
MatrizPontos[Pallet_1,Prdt_30All,4].NumCaixas = 4
MatrizPontos[Pallet_1,Prdt_30All,4].PickOp = 1
MatrizPontos[Pallet_1,Prdt_30All,4].ConfGarraOp = 0
MatrizPontos[Pallet_1,Prdt_30All,4].FechaGarraOp = 0
MatrizPontos[Pallet_1,Prdt_30All,4].AbreGarraOp = 0
MatrizPontos[Pallet_1,Prdt_30All,4].SensoresCaixa = 12345
MatrizPontos[Pallet_1,Prdt_30All,4].TravaGarra = False
MatrizPontos[Pallet_1,Prdt_30All,4].SkipGoHome = False
MatrizPontos[Pallet_1,Prdt_30All,4].SkipSobeRelAtual = False
MatrizPontos[Pallet_1,Prdt_30All,4].XApp1Place=P1_30All_4_App1
MatrizPontos[Pallet_1,Prdt_30All,4].XApp2Place=P1_30All_4_App2
MatrizPontos[Pallet_1,Prdt_30All,4].XPlace=P1_30All_4_Place
;ENDFOLD
;FOLD OffsetPlace
MatrizPontos[Pallet_1,Prdt_30All,4].OffsetPlace.X=0
MatrizPontos[Pallet_1,Prdt_30All,4].OffsetPlace.Y=0
MatrizPontos[Pallet_1,Prdt_30All,4].OffsetPlace.Z=0
MatrizPontos[Pallet_1,Prdt_30All,4].OffsetPlace.A=0
MatrizPontos[Pallet_1,Prdt_30All,4].OffsetPlace.B=0
MatrizPontos[Pallet_1,Prdt_30All,4].OffsetPlace.C=0
;ENDFOLD
;ENDFOLD

;ENDFOLD
;ENDFOLD

;FOLD Pallet 1 - Produto 16CoffeCrisp
;FOLD LAYER 1: PLACE 1 ate 4
;FOLD PLACE 1
;FOLD PROPRIEDADES
MatrizPontos[Pallet_1,Prdt_16CoffeCrisp,1].NumCaixas = 2
MatrizPontos[Pallet_1,Prdt_16CoffeCrisp,1].PickOp = 1
MatrizPontos[Pallet_1,Prdt_16CoffeCrisp,1].ConfGarraOp = 0
MatrizPontos[Pallet_1,Prdt_16CoffeCrisp,1].FechaGarraOp = 0
MatrizPontos[Pallet_1,Prdt_16CoffeCrisp,1].AbreGarraOp = 0
MatrizPontos[Pallet_1,Prdt_16CoffeCrisp,1].SensoresCaixa = 123
MatrizPontos[Pallet_1,Prdt_16CoffeCrisp,1].TravaGarra = False
MatrizPontos[Pallet_1,Prdt_16CoffeCrisp,1].SkipGoHome = False
MatrizPontos[Pallet_1,Prdt_16CoffeCrisp,1].SkipSobeRelAtual = False
MatrizPontos[Pallet_1,Prdt_16CoffeCrisp,1].XApp1Place=P1_16CoffeCrisp_1_App1
MatrizPontos[Pallet_1,Prdt_16CoffeCrisp,1].XApp2Place=P1_16CoffeCrisp_1_App2
MatrizPontos[Pallet_1,Prdt_16CoffeCrisp,1].XPlace=P1_16CoffeCrisp_1_Place
;ENDFOLD
;FOLD OffsetPlace
MatrizPontos[Pallet_1,Prdt_16CoffeCrisp,1].OffsetPlace.X=0
MatrizPontos[Pallet_1,Prdt_16CoffeCrisp,1].OffsetPlace.Y=0
MatrizPontos[Pallet_1,Prdt_16CoffeCrisp,1].OffsetPlace.Z=0
MatrizPontos[Pallet_1,Prdt_16CoffeCrisp,1].OffsetPlace.A=0
MatrizPontos[Pallet_1,Prdt_16CoffeCrisp,1].OffsetPlace.B=0
MatrizPontos[Pallet_1,Prdt_16CoffeCrisp,1].OffsetPlace.C=0
;ENDFOLD
;ENDFOLD

;FOLD PLACE 2
;FOLD PROPRIEDADES
MatrizPontos[Pallet_1,Prdt_16CoffeCrisp,2].NumCaixas = 2
MatrizPontos[Pallet_1,Prdt_16CoffeCrisp,2].PickOp = 1
MatrizPontos[Pallet_1,Prdt_16CoffeCrisp,2].ConfGarraOp = 0
MatrizPontos[Pallet_1,Prdt_16CoffeCrisp,2].FechaGarraOp = 0
MatrizPontos[Pallet_1,Prdt_16CoffeCrisp,2].AbreGarraOp = 0
MatrizPontos[Pallet_1,Prdt_16CoffeCrisp,2].SensoresCaixa = 123
MatrizPontos[Pallet_1,Prdt_16CoffeCrisp,2].TravaGarra = False
MatrizPontos[Pallet_1,Prdt_16CoffeCrisp,2].SkipGoHome = False
MatrizPontos[Pallet_1,Prdt_16CoffeCrisp,2].SkipSobeRelAtual = False
MatrizPontos[Pallet_1,Prdt_16CoffeCrisp,2].XApp1Place=P1_16CoffeCrisp_2_App1
MatrizPontos[Pallet_1,Prdt_16CoffeCrisp,2].XApp2Place=P1_16CoffeCrisp_2_App2
MatrizPontos[Pallet_1,Prdt_16CoffeCrisp,2].XPlace=P1_16CoffeCrisp_2_Place
;ENDFOLD
;FOLD OffsetPlace
MatrizPontos[Pallet_1,Prdt_16CoffeCrisp,2].OffsetPlace.X=0
MatrizPontos[Pallet_1,Prdt_16CoffeCrisp,2].OffsetPlace.Y=0
MatrizPontos[Pallet_1,Prdt_16CoffeCrisp,2].OffsetPlace.Z=0
MatrizPontos[Pallet_1,Prdt_16CoffeCrisp,2].OffsetPlace.A=0
MatrizPontos[Pallet_1,Prdt_16CoffeCrisp,2].OffsetPlace.B=0
MatrizPontos[Pallet_1,Prdt_16CoffeCrisp,2].OffsetPlace.C=0
;ENDFOLD
;ENDFOLD

;FOLD PLACE 3
;FOLD PROPRIEDADES
MatrizPontos[Pallet_1,Prdt_16CoffeCrisp,3].NumCaixas = 2
MatrizPontos[Pallet_1,Prdt_16CoffeCrisp,3].PickOp = 1
MatrizPontos[Pallet_1,Prdt_16CoffeCrisp,3].ConfGarraOp = 0
MatrizPontos[Pallet_1,Prdt_16CoffeCrisp,3].FechaGarraOp = 0
MatrizPontos[Pallet_1,Prdt_16CoffeCrisp,3].AbreGarraOp = 0
MatrizPontos[Pallet_1,Prdt_16CoffeCrisp,3].SensoresCaixa = 123
MatrizPontos[Pallet_1,Prdt_16CoffeCrisp,3].TravaGarra = False
MatrizPontos[Pallet_1,Prdt_16CoffeCrisp,3].SkipGoHome = False
MatrizPontos[Pallet_1,Prdt_16CoffeCrisp,3].SkipSobeRelAtual = False
MatrizPontos[Pallet_1,Prdt_16CoffeCrisp,3].XApp1Place=P1_16CoffeCrisp_3_App1
MatrizPontos[Pallet_1,Prdt_16CoffeCrisp,3].XApp2Place=P1_16CoffeCrisp_3_App2
MatrizPontos[Pallet_1,Prdt_16CoffeCrisp,3].XPlace=P1_16CoffeCrisp_3_Place
;ENDFOLD
;FOLD OffsetPlace
MatrizPontos[Pallet_1,Prdt_16CoffeCrisp,3].OffsetPlace.X=0
MatrizPontos[Pallet_1,Prdt_16CoffeCrisp,3].OffsetPlace.Y=0
MatrizPontos[Pallet_1,Prdt_16CoffeCrisp,3].OffsetPlace.Z=0
MatrizPontos[Pallet_1,Prdt_16CoffeCrisp,3].OffsetPlace.A=0
MatrizPontos[Pallet_1,Prdt_16CoffeCrisp,3].OffsetPlace.B=0
MatrizPontos[Pallet_1,Prdt_16CoffeCrisp,3].OffsetPlace.C=0
;ENDFOLD
;ENDFOLD

;FOLD PLACE 4
;FOLD PROPRIEDADES
MatrizPontos[Pallet_1,Prdt_16CoffeCrisp,4].NumCaixas = 4
MatrizPontos[Pallet_1,Prdt_16CoffeCrisp,4].PickOp = 1
MatrizPontos[Pallet_1,Prdt_16CoffeCrisp,4].ConfGarraOp = 0
MatrizPontos[Pallet_1,Prdt_16CoffeCrisp,4].FechaGarraOp = 0
MatrizPontos[Pallet_1,Prdt_16CoffeCrisp,4].AbreGarraOp = 0
MatrizPontos[Pallet_1,Prdt_16CoffeCrisp,4].SensoresCaixa = 123456
MatrizPontos[Pallet_1,Prdt_16CoffeCrisp,4].TravaGarra = False
MatrizPontos[Pallet_1,Prdt_16CoffeCrisp,4].SkipGoHome = False
MatrizPontos[Pallet_1,Prdt_16CoffeCrisp,4].SkipSobeRelAtual = False
MatrizPontos[Pallet_1,Prdt_16CoffeCrisp,4].XApp1Place=P1_16CoffeCrisp_4_App1
MatrizPontos[Pallet_1,Prdt_16CoffeCrisp,4].XApp2Place=P1_16CoffeCrisp_4_App2
MatrizPontos[Pallet_1,Prdt_16CoffeCrisp,4].XPlace=P1_16CoffeCrisp_4_Place
;ENDFOLD
;FOLD OffsetPlace
MatrizPontos[Pallet_1,Prdt_16CoffeCrisp,4].OffsetPlace.X=0
MatrizPontos[Pallet_1,Prdt_16CoffeCrisp,4].OffsetPlace.Y=0
MatrizPontos[Pallet_1,Prdt_16CoffeCrisp,4].OffsetPlace.Z=0
MatrizPontos[Pallet_1,Prdt_16CoffeCrisp,4].OffsetPlace.A=0
MatrizPontos[Pallet_1,Prdt_16CoffeCrisp,4].OffsetPlace.B=0
MatrizPontos[Pallet_1,Prdt_16CoffeCrisp,4].OffsetPlace.C=0
;ENDFOLD
;ENDFOLD

;ENDFOLD
;FOLD LAYER 2: PLACE 5 ate 8
;FOLD PLACE 5
;FOLD PROPRIEDADES
MatrizPontos[Pallet_1,Prdt_16CoffeCrisp,5].NumCaixas = 4
MatrizPontos[Pallet_1,Prdt_16CoffeCrisp,5].PickOp = 1
MatrizPontos[Pallet_1,Prdt_16CoffeCrisp,5].ConfGarraOp = 0
MatrizPontos[Pallet_1,Prdt_16CoffeCrisp,5].FechaGarraOp = 0
MatrizPontos[Pallet_1,Prdt_16CoffeCrisp,5].AbreGarraOp = 0
MatrizPontos[Pallet_1,Prdt_16CoffeCrisp,5].SensoresCaixa = 123456
MatrizPontos[Pallet_1,Prdt_16CoffeCrisp,5].TravaGarra = False
MatrizPontos[Pallet_1,Prdt_16CoffeCrisp,5].SkipGoHome = False
MatrizPontos[Pallet_1,Prdt_16CoffeCrisp,5].SkipSobeRelAtual = False
MatrizPontos[Pallet_1,Prdt_16CoffeCrisp,5].XApp1Place=P1_16CoffeCrisp_5_App1
MatrizPontos[Pallet_1,Prdt_16CoffeCrisp,5].XApp2Place=P1_16CoffeCrisp_5_App2
MatrizPontos[Pallet_1,Prdt_16CoffeCrisp,5].XPlace=P1_16CoffeCrisp_5_Place
;ENDFOLD
;FOLD OffsetPlace
MatrizPontos[Pallet_1,Prdt_16CoffeCrisp,5].OffsetPlace.X=0
MatrizPontos[Pallet_1,Prdt_16CoffeCrisp,5].OffsetPlace.Y=0
MatrizPontos[Pallet_1,Prdt_16CoffeCrisp,5].OffsetPlace.Z=0
MatrizPontos[Pallet_1,Prdt_16CoffeCrisp,5].OffsetPlace.A=0
MatrizPontos[Pallet_1,Prdt_16CoffeCrisp,5].OffsetPlace.B=0
MatrizPontos[Pallet_1,Prdt_16CoffeCrisp,5].OffsetPlace.C=0
;ENDFOLD
;ENDFOLD

;FOLD PLACE 6
;FOLD PROPRIEDADES
MatrizPontos[Pallet_1,Prdt_16CoffeCrisp,6].NumCaixas = 2
MatrizPontos[Pallet_1,Prdt_16CoffeCrisp,6].PickOp = 1
MatrizPontos[Pallet_1,Prdt_16CoffeCrisp,6].ConfGarraOp = 0
MatrizPontos[Pallet_1,Prdt_16CoffeCrisp,6].FechaGarraOp = 0
MatrizPontos[Pallet_1,Prdt_16CoffeCrisp,6].AbreGarraOp = 0
MatrizPontos[Pallet_1,Prdt_16CoffeCrisp,6].SensoresCaixa = 123
MatrizPontos[Pallet_1,Prdt_16CoffeCrisp,6].TravaGarra = False
MatrizPontos[Pallet_1,Prdt_16CoffeCrisp,6].SkipGoHome = False
MatrizPontos[Pallet_1,Prdt_16CoffeCrisp,6].SkipSobeRelAtual = False
MatrizPontos[Pallet_1,Prdt_16CoffeCrisp,6].XApp1Place=P1_16CoffeCrisp_6_App1
MatrizPontos[Pallet_1,Prdt_16CoffeCrisp,6].XApp2Place=P1_16CoffeCrisp_6_App2
MatrizPontos[Pallet_1,Prdt_16CoffeCrisp,6].XPlace=P1_16CoffeCrisp_6_Place
;ENDFOLD
;FOLD OffsetPlace
MatrizPontos[Pallet_1,Prdt_16CoffeCrisp,6].OffsetPlace.X=0
MatrizPontos[Pallet_1,Prdt_16CoffeCrisp,6].OffsetPlace.Y=0
MatrizPontos[Pallet_1,Prdt_16CoffeCrisp,6].OffsetPlace.Z=0
MatrizPontos[Pallet_1,Prdt_16CoffeCrisp,6].OffsetPlace.A=0
MatrizPontos[Pallet_1,Prdt_16CoffeCrisp,6].OffsetPlace.B=0
MatrizPontos[Pallet_1,Prdt_16CoffeCrisp,6].OffsetPlace.C=0
;ENDFOLD
;ENDFOLD

;FOLD PLACE 7
;FOLD PROPRIEDADES
MatrizPontos[Pallet_1,Prdt_16CoffeCrisp,7].NumCaixas = 2
MatrizPontos[Pallet_1,Prdt_16CoffeCrisp,7].PickOp = 1
MatrizPontos[Pallet_1,Prdt_16CoffeCrisp,7].ConfGarraOp = 0
MatrizPontos[Pallet_1,Prdt_16CoffeCrisp,7].FechaGarraOp = 0
MatrizPontos[Pallet_1,Prdt_16CoffeCrisp,7].AbreGarraOp = 0
MatrizPontos[Pallet_1,Prdt_16CoffeCrisp,7].SensoresCaixa = 123
MatrizPontos[Pallet_1,Prdt_16CoffeCrisp,7].TravaGarra = False
MatrizPontos[Pallet_1,Prdt_16CoffeCrisp,7].SkipGoHome = False
MatrizPontos[Pallet_1,Prdt_16CoffeCrisp,7].SkipSobeRelAtual = False
MatrizPontos[Pallet_1,Prdt_16CoffeCrisp,7].XApp1Place=P1_16CoffeCrisp_7_App1
MatrizPontos[Pallet_1,Prdt_16CoffeCrisp,7].XApp2Place=P1_16CoffeCrisp_7_App2
MatrizPontos[Pallet_1,Prdt_16CoffeCrisp,7].XPlace=P1_16CoffeCrisp_7_Place
;ENDFOLD
;FOLD OffsetPlace
MatrizPontos[Pallet_1,Prdt_16CoffeCrisp,7].OffsetPlace.X=0
MatrizPontos[Pallet_1,Prdt_16CoffeCrisp,7].OffsetPlace.Y=0
MatrizPontos[Pallet_1,Prdt_16CoffeCrisp,7].OffsetPlace.Z=0
MatrizPontos[Pallet_1,Prdt_16CoffeCrisp,7].OffsetPlace.A=0
MatrizPontos[Pallet_1,Prdt_16CoffeCrisp,7].OffsetPlace.B=0
MatrizPontos[Pallet_1,Prdt_16CoffeCrisp,7].OffsetPlace.C=0
;ENDFOLD
;ENDFOLD

;FOLD PLACE 8
;FOLD PROPRIEDADES
MatrizPontos[Pallet_1,Prdt_16CoffeCrisp,8].NumCaixas = 2
MatrizPontos[Pallet_1,Prdt_16CoffeCrisp,8].PickOp = 1
MatrizPontos[Pallet_1,Prdt_16CoffeCrisp,8].ConfGarraOp = 0
MatrizPontos[Pallet_1,Prdt_16CoffeCrisp,8].FechaGarraOp = 0
MatrizPontos[Pallet_1,Prdt_16CoffeCrisp,8].AbreGarraOp = 0
MatrizPontos[Pallet_1,Prdt_16CoffeCrisp,8].SensoresCaixa = 123
MatrizPontos[Pallet_1,Prdt_16CoffeCrisp,8].TravaGarra = False
MatrizPontos[Pallet_1,Prdt_16CoffeCrisp,8].SkipGoHome = False
MatrizPontos[Pallet_1,Prdt_16CoffeCrisp,8].SkipSobeRelAtual = False
MatrizPontos[Pallet_1,Prdt_16CoffeCrisp,8].XApp1Place=P1_16CoffeCrisp_8_App1
MatrizPontos[Pallet_1,Prdt_16CoffeCrisp,8].XApp2Place=P1_16CoffeCrisp_8_App2
MatrizPontos[Pallet_1,Prdt_16CoffeCrisp,8].XPlace=P1_16CoffeCrisp_8_Place
;ENDFOLD
;FOLD OffsetPlace
MatrizPontos[Pallet_1,Prdt_16CoffeCrisp,8].OffsetPlace.X=0
MatrizPontos[Pallet_1,Prdt_16CoffeCrisp,8].OffsetPlace.Y=0
MatrizPontos[Pallet_1,Prdt_16CoffeCrisp,8].OffsetPlace.Z=0
MatrizPontos[Pallet_1,Prdt_16CoffeCrisp,8].OffsetPlace.A=0
MatrizPontos[Pallet_1,Prdt_16CoffeCrisp,8].OffsetPlace.B=0
MatrizPontos[Pallet_1,Prdt_16CoffeCrisp,8].OffsetPlace.C=0
;ENDFOLD
;ENDFOLD

;ENDFOLD
;ENDFOLD

;FOLD Pallet 1 - Produto 10CoffeCrisp
;FOLD LAYER 1: PLACE 1 ate 4
;FOLD PLACE 1
;FOLD PROPRIEDADES
MatrizPontos[Pallet_1,Prdt_10CoffeCrisp,1].NumCaixas = 1
MatrizPontos[Pallet_1,Prdt_10CoffeCrisp,1].PickOp = 6
MatrizPontos[Pallet_1,Prdt_10CoffeCrisp,1].ConfGarraOp = 0
MatrizPontos[Pallet_1,Prdt_10CoffeCrisp,1].FechaGarraOp = 0
MatrizPontos[Pallet_1,Prdt_10CoffeCrisp,1].AbreGarraOp = 0
MatrizPontos[Pallet_1,Prdt_10CoffeCrisp,1].SensoresCaixa = 56
MatrizPontos[Pallet_1,Prdt_10CoffeCrisp,1].TravaGarra = False
MatrizPontos[Pallet_1,Prdt_10CoffeCrisp,1].SkipGoHome = False
MatrizPontos[Pallet_1,Prdt_10CoffeCrisp,1].SkipSobeRelAtual = False
MatrizPontos[Pallet_1,Prdt_10CoffeCrisp,1].XApp1Place=P1_10CoffeCrisp_1_App1
MatrizPontos[Pallet_1,Prdt_10CoffeCrisp,1].XApp2Place=P1_10CoffeCrisp_1_App2
MatrizPontos[Pallet_1,Prdt_10CoffeCrisp,1].XPlace=P1_10CoffeCrisp_1_Place
;ENDFOLD
;FOLD OffsetPlace
MatrizPontos[Pallet_1,Prdt_10CoffeCrisp,1].OffsetPlace.X=0
MatrizPontos[Pallet_1,Prdt_10CoffeCrisp,1].OffsetPlace.Y=0
MatrizPontos[Pallet_1,Prdt_10CoffeCrisp,1].OffsetPlace.Z=0
MatrizPontos[Pallet_1,Prdt_10CoffeCrisp,1].OffsetPlace.A=0
MatrizPontos[Pallet_1,Prdt_10CoffeCrisp,1].OffsetPlace.B=0
MatrizPontos[Pallet_1,Prdt_10CoffeCrisp,1].OffsetPlace.C=0
;ENDFOLD
;ENDFOLD

;FOLD PLACE 2
;FOLD PROPRIEDADES
MatrizPontos[Pallet_1,Prdt_10CoffeCrisp,2].NumCaixas = 1
MatrizPontos[Pallet_1,Prdt_10CoffeCrisp,2].PickOp = 6
MatrizPontos[Pallet_1,Prdt_10CoffeCrisp,2].ConfGarraOp = 0
MatrizPontos[Pallet_1,Prdt_10CoffeCrisp,2].FechaGarraOp = 0
MatrizPontos[Pallet_1,Prdt_10CoffeCrisp,2].AbreGarraOp = 0
MatrizPontos[Pallet_1,Prdt_10CoffeCrisp,2].SensoresCaixa = 56
MatrizPontos[Pallet_1,Prdt_10CoffeCrisp,2].TravaGarra = False
MatrizPontos[Pallet_1,Prdt_10CoffeCrisp,2].SkipGoHome = False
MatrizPontos[Pallet_1,Prdt_10CoffeCrisp,2].SkipSobeRelAtual = False
MatrizPontos[Pallet_1,Prdt_10CoffeCrisp,2].XApp1Place=P1_10CoffeCrisp_2_App1
MatrizPontos[Pallet_1,Prdt_10CoffeCrisp,2].XApp2Place=P1_10CoffeCrisp_2_App2
MatrizPontos[Pallet_1,Prdt_10CoffeCrisp,2].XPlace=P1_10CoffeCrisp_2_Place
;ENDFOLD
;FOLD OffsetPlace
MatrizPontos[Pallet_1,Prdt_10CoffeCrisp,2].OffsetPlace.X=0
MatrizPontos[Pallet_1,Prdt_10CoffeCrisp,2].OffsetPlace.Y=0
MatrizPontos[Pallet_1,Prdt_10CoffeCrisp,2].OffsetPlace.Z=0
MatrizPontos[Pallet_1,Prdt_10CoffeCrisp,2].OffsetPlace.A=0
MatrizPontos[Pallet_1,Prdt_10CoffeCrisp,2].OffsetPlace.B=0
MatrizPontos[Pallet_1,Prdt_10CoffeCrisp,2].OffsetPlace.C=0
;ENDFOLD
;ENDFOLD

;FOLD PLACE 3
;FOLD PROPRIEDADES
MatrizPontos[Pallet_1,Prdt_10CoffeCrisp,3].NumCaixas = 3
MatrizPontos[Pallet_1,Prdt_10CoffeCrisp,3].PickOp = 1
MatrizPontos[Pallet_1,Prdt_10CoffeCrisp,3].ConfGarraOp = 0
MatrizPontos[Pallet_1,Prdt_10CoffeCrisp,3].FechaGarraOp = 0
MatrizPontos[Pallet_1,Prdt_10CoffeCrisp,3].AbreGarraOp = 0
MatrizPontos[Pallet_1,Prdt_10CoffeCrisp,3].SensoresCaixa = 12345
MatrizPontos[Pallet_1,Prdt_10CoffeCrisp,3].TravaGarra = False
MatrizPontos[Pallet_1,Prdt_10CoffeCrisp,3].SkipGoHome = False
MatrizPontos[Pallet_1,Prdt_10CoffeCrisp,3].SkipSobeRelAtual = False
MatrizPontos[Pallet_1,Prdt_10CoffeCrisp,3].XApp1Place=P1_10CoffeCrisp_3_App1
MatrizPontos[Pallet_1,Prdt_10CoffeCrisp,3].XApp2Place=P1_10CoffeCrisp_3_App2
MatrizPontos[Pallet_1,Prdt_10CoffeCrisp,3].XPlace=P1_10CoffeCrisp_3_Place
;ENDFOLD
;FOLD OffsetPlace
MatrizPontos[Pallet_1,Prdt_10CoffeCrisp,3].OffsetPlace.X=0
MatrizPontos[Pallet_1,Prdt_10CoffeCrisp,3].OffsetPlace.Y=0
MatrizPontos[Pallet_1,Prdt_10CoffeCrisp,3].OffsetPlace.Z=0
MatrizPontos[Pallet_1,Prdt_10CoffeCrisp,3].OffsetPlace.A=0
MatrizPontos[Pallet_1,Prdt_10CoffeCrisp,3].OffsetPlace.B=0
MatrizPontos[Pallet_1,Prdt_10CoffeCrisp,3].OffsetPlace.C=0
;ENDFOLD
;ENDFOLD

;FOLD PLACE 4
;FOLD PROPRIEDADES
MatrizPontos[Pallet_1,Prdt_10CoffeCrisp,4].NumCaixas = 3
MatrizPontos[Pallet_1,Prdt_10CoffeCrisp,4].PickOp = 1
MatrizPontos[Pallet_1,Prdt_10CoffeCrisp,4].ConfGarraOp = 0
MatrizPontos[Pallet_1,Prdt_10CoffeCrisp,4].FechaGarraOp = 0
MatrizPontos[Pallet_1,Prdt_10CoffeCrisp,4].AbreGarraOp = 0
MatrizPontos[Pallet_1,Prdt_10CoffeCrisp,4].SensoresCaixa = 12345
MatrizPontos[Pallet_1,Prdt_10CoffeCrisp,4].TravaGarra = False
MatrizPontos[Pallet_1,Prdt_10CoffeCrisp,4].SkipGoHome = False
MatrizPontos[Pallet_1,Prdt_10CoffeCrisp,4].SkipSobeRelAtual = False
MatrizPontos[Pallet_1,Prdt_10CoffeCrisp,4].XApp1Place=P1_10CoffeCrisp_4_App1
MatrizPontos[Pallet_1,Prdt_10CoffeCrisp,4].XApp2Place=P1_10CoffeCrisp_4_App2
MatrizPontos[Pallet_1,Prdt_10CoffeCrisp,4].XPlace=P1_10CoffeCrisp_4_Place
;ENDFOLD
;FOLD OffsetPlace
MatrizPontos[Pallet_1,Prdt_10CoffeCrisp,4].OffsetPlace.X=0
MatrizPontos[Pallet_1,Prdt_10CoffeCrisp,4].OffsetPlace.Y=0
MatrizPontos[Pallet_1,Prdt_10CoffeCrisp,4].OffsetPlace.Z=0
MatrizPontos[Pallet_1,Prdt_10CoffeCrisp,4].OffsetPlace.A=0
MatrizPontos[Pallet_1,Prdt_10CoffeCrisp,4].OffsetPlace.B=0
MatrizPontos[Pallet_1,Prdt_10CoffeCrisp,4].OffsetPlace.C=0
;ENDFOLD
;ENDFOLD

;ENDFOLD
;FOLD LAYER 2: PLACE 5 ate 8
;FOLD PLACE 5
;FOLD PROPRIEDADES
MatrizPontos[Pallet_1,Prdt_10CoffeCrisp,5].NumCaixas = 1
MatrizPontos[Pallet_1,Prdt_10CoffeCrisp,5].PickOp = 3
MatrizPontos[Pallet_1,Prdt_10CoffeCrisp,5].ConfGarraOp = 3
MatrizPontos[Pallet_1,Prdt_10CoffeCrisp,5].FechaGarraOp = 0
MatrizPontos[Pallet_1,Prdt_10CoffeCrisp,5].AbreGarraOp = 0
MatrizPontos[Pallet_1,Prdt_10CoffeCrisp,5].SensoresCaixa = 12
MatrizPontos[Pallet_1,Prdt_10CoffeCrisp,5].TravaGarra = False
MatrizPontos[Pallet_1,Prdt_10CoffeCrisp,5].SkipGoHome = False
MatrizPontos[Pallet_1,Prdt_10CoffeCrisp,5].SkipSobeRelAtual = False
MatrizPontos[Pallet_1,Prdt_10CoffeCrisp,5].XApp1Place=P1_10CoffeCrisp_5_App1
MatrizPontos[Pallet_1,Prdt_10CoffeCrisp,5].XApp2Place=P1_10CoffeCrisp_5_App2
MatrizPontos[Pallet_1,Prdt_10CoffeCrisp,5].XPlace=P1_10CoffeCrisp_5_Place
;ENDFOLD
;FOLD OffsetPlace
MatrizPontos[Pallet_1,Prdt_10CoffeCrisp,5].OffsetPlace.X=0
MatrizPontos[Pallet_1,Prdt_10CoffeCrisp,5].OffsetPlace.Y=0
MatrizPontos[Pallet_1,Prdt_10CoffeCrisp,5].OffsetPlace.Z=0
MatrizPontos[Pallet_1,Prdt_10CoffeCrisp,5].OffsetPlace.A=0
MatrizPontos[Pallet_1,Prdt_10CoffeCrisp,5].OffsetPlace.B=0
MatrizPontos[Pallet_1,Prdt_10CoffeCrisp,5].OffsetPlace.C=0
;ENDFOLD
;ENDFOLD

;FOLD PLACE 6
;FOLD PROPRIEDADES
MatrizPontos[Pallet_1,Prdt_10CoffeCrisp,6].NumCaixas = 1
MatrizPontos[Pallet_1,Prdt_10CoffeCrisp,6].PickOp = 3
MatrizPontos[Pallet_1,Prdt_10CoffeCrisp,6].ConfGarraOp = 3
MatrizPontos[Pallet_1,Prdt_10CoffeCrisp,6].FechaGarraOp = 0
MatrizPontos[Pallet_1,Prdt_10CoffeCrisp,6].AbreGarraOp = 0
MatrizPontos[Pallet_1,Prdt_10CoffeCrisp,6].SensoresCaixa = 12
MatrizPontos[Pallet_1,Prdt_10CoffeCrisp,6].TravaGarra = False
MatrizPontos[Pallet_1,Prdt_10CoffeCrisp,6].SkipGoHome = False
MatrizPontos[Pallet_1,Prdt_10CoffeCrisp,6].SkipSobeRelAtual = False
MatrizPontos[Pallet_1,Prdt_10CoffeCrisp,6].XApp1Place=P1_10CoffeCrisp_6_App1
MatrizPontos[Pallet_1,Prdt_10CoffeCrisp,6].XApp2Place=P1_10CoffeCrisp_6_App2
MatrizPontos[Pallet_1,Prdt_10CoffeCrisp,6].XPlace=P1_10CoffeCrisp_6_Place
;ENDFOLD
;FOLD OffsetPlace
MatrizPontos[Pallet_1,Prdt_10CoffeCrisp,6].OffsetPlace.X=0
MatrizPontos[Pallet_1,Prdt_10CoffeCrisp,6].OffsetPlace.Y=0
MatrizPontos[Pallet_1,Prdt_10CoffeCrisp,6].OffsetPlace.Z=0
MatrizPontos[Pallet_1,Prdt_10CoffeCrisp,6].OffsetPlace.A=0
MatrizPontos[Pallet_1,Prdt_10CoffeCrisp,6].OffsetPlace.B=0
MatrizPontos[Pallet_1,Prdt_10CoffeCrisp,6].OffsetPlace.C=0
;ENDFOLD
;ENDFOLD

;FOLD PLACE 7
;FOLD PROPRIEDADES
MatrizPontos[Pallet_1,Prdt_10CoffeCrisp,7].NumCaixas = 3
MatrizPontos[Pallet_1,Prdt_10CoffeCrisp,7].PickOp = 1
MatrizPontos[Pallet_1,Prdt_10CoffeCrisp,7].ConfGarraOp = 0
MatrizPontos[Pallet_1,Prdt_10CoffeCrisp,7].FechaGarraOp = 0
MatrizPontos[Pallet_1,Prdt_10CoffeCrisp,7].AbreGarraOp = 1
MatrizPontos[Pallet_1,Prdt_10CoffeCrisp,7].SensoresCaixa = 12345
MatrizPontos[Pallet_1,Prdt_10CoffeCrisp,7].TravaGarra = True
MatrizPontos[Pallet_1,Prdt_10CoffeCrisp,7].SkipGoHome = False
MatrizPontos[Pallet_1,Prdt_10CoffeCrisp,7].SkipSobeRelAtual = False
MatrizPontos[Pallet_1,Prdt_10CoffeCrisp,7].XApp1Place=P1_10CoffeCrisp_7_App1
MatrizPontos[Pallet_1,Prdt_10CoffeCrisp,7].XApp2Place=P1_10CoffeCrisp_7_App2
MatrizPontos[Pallet_1,Prdt_10CoffeCrisp,7].XPlace=P1_10CoffeCrisp_7_Place
;ENDFOLD
;FOLD OffsetPlace
MatrizPontos[Pallet_1,Prdt_10CoffeCrisp,7].OffsetPlace.X=0
MatrizPontos[Pallet_1,Prdt_10CoffeCrisp,7].OffsetPlace.Y=0
MatrizPontos[Pallet_1,Prdt_10CoffeCrisp,7].OffsetPlace.Z=0
MatrizPontos[Pallet_1,Prdt_10CoffeCrisp,7].OffsetPlace.A=0
MatrizPontos[Pallet_1,Prdt_10CoffeCrisp,7].OffsetPlace.B=0
MatrizPontos[Pallet_1,Prdt_10CoffeCrisp,7].OffsetPlace.C=0
;ENDFOLD
;ENDFOLD

;FOLD PLACE 8
;FOLD PROPRIEDADES
MatrizPontos[Pallet_1,Prdt_10CoffeCrisp,8].NumCaixas = 3
MatrizPontos[Pallet_1,Prdt_10CoffeCrisp,8].PickOp = 1
MatrizPontos[Pallet_1,Prdt_10CoffeCrisp,8].ConfGarraOp = 0
MatrizPontos[Pallet_1,Prdt_10CoffeCrisp,8].FechaGarraOp = 0
MatrizPontos[Pallet_1,Prdt_10CoffeCrisp,8].AbreGarraOp = 1
MatrizPontos[Pallet_1,Prdt_10CoffeCrisp,8].SensoresCaixa = 12345
MatrizPontos[Pallet_1,Prdt_10CoffeCrisp,8].TravaGarra = True
MatrizPontos[Pallet_1,Prdt_10CoffeCrisp,8].SkipGoHome = False
MatrizPontos[Pallet_1,Prdt_10CoffeCrisp,8].SkipSobeRelAtual = False
MatrizPontos[Pallet_1,Prdt_10CoffeCrisp,8].XApp1Place=P1_10CoffeCrisp_8_App1
MatrizPontos[Pallet_1,Prdt_10CoffeCrisp,8].XApp2Place=P1_10CoffeCrisp_8_App2
MatrizPontos[Pallet_1,Prdt_10CoffeCrisp,8].XPlace=P1_10CoffeCrisp_8_Place
;ENDFOLD
;FOLD OffsetPlace
MatrizPontos[Pallet_1,Prdt_10CoffeCrisp,8].OffsetPlace.X=0
MatrizPontos[Pallet_1,Prdt_10CoffeCrisp,8].OffsetPlace.Y=0
MatrizPontos[Pallet_1,Prdt_10CoffeCrisp,8].OffsetPlace.Z=0
MatrizPontos[Pallet_1,Prdt_10CoffeCrisp,8].OffsetPlace.A=0
MatrizPontos[Pallet_1,Prdt_10CoffeCrisp,8].OffsetPlace.B=0
MatrizPontos[Pallet_1,Prdt_10CoffeCrisp,8].OffsetPlace.C=0
;ENDFOLD
;ENDFOLD

;ENDFOLD
;ENDFOLD

;FOLD Pallet 1 - Produto 15CoffeCrisp
;FOLD LAYER 1: PLACE 1 ate 7
;FOLD PLACE 1
;FOLD PROPRIEDADES
MatrizPontos[Pallet_1,Prdt_15CoffeCrisp,1].NumCaixas = 1
MatrizPontos[Pallet_1,Prdt_15CoffeCrisp,1].PickOp = 8
MatrizPontos[Pallet_1,Prdt_15CoffeCrisp,1].ConfGarraOp = 5
MatrizPontos[Pallet_1,Prdt_15CoffeCrisp,1].FechaGarraOp = 0
MatrizPontos[Pallet_1,Prdt_15CoffeCrisp,1].AbreGarraOp = 0
MatrizPontos[Pallet_1,Prdt_15CoffeCrisp,1].SensoresCaixa = 1
MatrizPontos[Pallet_1,Prdt_15CoffeCrisp,1].TravaGarra = False
MatrizPontos[Pallet_1,Prdt_15CoffeCrisp,1].SkipGoHome = False
MatrizPontos[Pallet_1,Prdt_15CoffeCrisp,1].SkipSobeRelAtual = False
MatrizPontos[Pallet_1,Prdt_15CoffeCrisp,1].XApp1Place=P1_15CoffeCrisp_1_App1
MatrizPontos[Pallet_1,Prdt_15CoffeCrisp,1].XApp2Place=P1_15CoffeCrisp_1_App2
MatrizPontos[Pallet_1,Prdt_15CoffeCrisp,1].XPlace=P1_15CoffeCrisp_1_Place
;ENDFOLD
;FOLD OffsetPlace
MatrizPontos[Pallet_1,Prdt_15CoffeCrisp,1].OffsetPlace.X=0
MatrizPontos[Pallet_1,Prdt_15CoffeCrisp,1].OffsetPlace.Y=0
MatrizPontos[Pallet_1,Prdt_15CoffeCrisp,1].OffsetPlace.Z=0
MatrizPontos[Pallet_1,Prdt_15CoffeCrisp,1].OffsetPlace.A=0
MatrizPontos[Pallet_1,Prdt_15CoffeCrisp,1].OffsetPlace.B=0
MatrizPontos[Pallet_1,Prdt_15CoffeCrisp,1].OffsetPlace.C=0
;ENDFOLD
;ENDFOLD

;FOLD PLACE 2
;FOLD PROPRIEDADES
MatrizPontos[Pallet_1,Prdt_15CoffeCrisp,2].NumCaixas = 1
MatrizPontos[Pallet_1,Prdt_15CoffeCrisp,2].PickOp = 8
MatrizPontos[Pallet_1,Prdt_15CoffeCrisp,2].ConfGarraOp = 5
MatrizPontos[Pallet_1,Prdt_15CoffeCrisp,2].FechaGarraOp = 0
MatrizPontos[Pallet_1,Prdt_15CoffeCrisp,2].AbreGarraOp = 0
MatrizPontos[Pallet_1,Prdt_15CoffeCrisp,2].SensoresCaixa = 1
MatrizPontos[Pallet_1,Prdt_15CoffeCrisp,2].TravaGarra = False
MatrizPontos[Pallet_1,Prdt_15CoffeCrisp,2].SkipGoHome = False
MatrizPontos[Pallet_1,Prdt_15CoffeCrisp,2].SkipSobeRelAtual = False
MatrizPontos[Pallet_1,Prdt_15CoffeCrisp,2].XApp1Place=P1_15CoffeCrisp_2_App1
MatrizPontos[Pallet_1,Prdt_15CoffeCrisp,2].XApp2Place=P1_15CoffeCrisp_2_App2
MatrizPontos[Pallet_1,Prdt_15CoffeCrisp,2].XPlace=P1_15CoffeCrisp_2_Place
;ENDFOLD
;FOLD OffsetPlace
MatrizPontos[Pallet_1,Prdt_15CoffeCrisp,2].OffsetPlace.X=0
MatrizPontos[Pallet_1,Prdt_15CoffeCrisp,2].OffsetPlace.Y=0
MatrizPontos[Pallet_1,Prdt_15CoffeCrisp,2].OffsetPlace.Z=0
MatrizPontos[Pallet_1,Prdt_15CoffeCrisp,2].OffsetPlace.A=0
MatrizPontos[Pallet_1,Prdt_15CoffeCrisp,2].OffsetPlace.B=0
MatrizPontos[Pallet_1,Prdt_15CoffeCrisp,2].OffsetPlace.C=0
;ENDFOLD
;ENDFOLD

;FOLD PLACE 3
;FOLD PROPRIEDADES
MatrizPontos[Pallet_1,Prdt_15CoffeCrisp,3].NumCaixas = 1
MatrizPontos[Pallet_1,Prdt_15CoffeCrisp,3].PickOp = 8
MatrizPontos[Pallet_1,Prdt_15CoffeCrisp,3].ConfGarraOp = 5
MatrizPontos[Pallet_1,Prdt_15CoffeCrisp,3].FechaGarraOp = 0
MatrizPontos[Pallet_1,Prdt_15CoffeCrisp,3].AbreGarraOp = 0
MatrizPontos[Pallet_1,Prdt_15CoffeCrisp,3].SensoresCaixa = 1
MatrizPontos[Pallet_1,Prdt_15CoffeCrisp,3].TravaGarra = False
MatrizPontos[Pallet_1,Prdt_15CoffeCrisp,3].SkipGoHome = False
MatrizPontos[Pallet_1,Prdt_15CoffeCrisp,3].SkipSobeRelAtual = False
MatrizPontos[Pallet_1,Prdt_15CoffeCrisp,3].XApp1Place=P1_15CoffeCrisp_3_App1
MatrizPontos[Pallet_1,Prdt_15CoffeCrisp,3].XApp2Place=P1_15CoffeCrisp_3_App2
MatrizPontos[Pallet_1,Prdt_15CoffeCrisp,3].XPlace=P1_15CoffeCrisp_3_Place
;ENDFOLD
;FOLD OffsetPlace
MatrizPontos[Pallet_1,Prdt_15CoffeCrisp,3].OffsetPlace.X=0
MatrizPontos[Pallet_1,Prdt_15CoffeCrisp,3].OffsetPlace.Y=0
MatrizPontos[Pallet_1,Prdt_15CoffeCrisp,3].OffsetPlace.Z=0
MatrizPontos[Pallet_1,Prdt_15CoffeCrisp,3].OffsetPlace.A=0
MatrizPontos[Pallet_1,Prdt_15CoffeCrisp,3].OffsetPlace.B=0
MatrizPontos[Pallet_1,Prdt_15CoffeCrisp,3].OffsetPlace.C=0
;ENDFOLD
;ENDFOLD

;FOLD PLACE 4
;FOLD PROPRIEDADES
MatrizPontos[Pallet_1,Prdt_15CoffeCrisp,4].NumCaixas = 2
MatrizPontos[Pallet_1,Prdt_15CoffeCrisp,4].PickOp = 8
MatrizPontos[Pallet_1,Prdt_15CoffeCrisp,4].ConfGarraOp = 5
MatrizPontos[Pallet_1,Prdt_15CoffeCrisp,4].FechaGarraOp = 0
MatrizPontos[Pallet_1,Prdt_15CoffeCrisp,4].AbreGarraOp = 1
MatrizPontos[Pallet_1,Prdt_15CoffeCrisp,4].SensoresCaixa = 123
MatrizPontos[Pallet_1,Prdt_15CoffeCrisp,4].TravaGarra = True
MatrizPontos[Pallet_1,Prdt_15CoffeCrisp,4].SkipGoHome = False
MatrizPontos[Pallet_1,Prdt_15CoffeCrisp,4].SkipSobeRelAtual = False
MatrizPontos[Pallet_1,Prdt_15CoffeCrisp,4].XApp1Place=P1_15CoffeCrisp_4_App1
MatrizPontos[Pallet_1,Prdt_15CoffeCrisp,4].XApp2Place=P1_15CoffeCrisp_4_App2
MatrizPontos[Pallet_1,Prdt_15CoffeCrisp,4].XPlace=P1_15CoffeCrisp_4_Place
;ENDFOLD
;FOLD OffsetPlace
MatrizPontos[Pallet_1,Prdt_15CoffeCrisp,4].OffsetPlace.X=0
MatrizPontos[Pallet_1,Prdt_15CoffeCrisp,4].OffsetPlace.Y=0
MatrizPontos[Pallet_1,Prdt_15CoffeCrisp,4].OffsetPlace.Z=0
MatrizPontos[Pallet_1,Prdt_15CoffeCrisp,4].OffsetPlace.A=0
MatrizPontos[Pallet_1,Prdt_15CoffeCrisp,4].OffsetPlace.B=0
MatrizPontos[Pallet_1,Prdt_15CoffeCrisp,4].OffsetPlace.C=0
;ENDFOLD
;ENDFOLD

;FOLD PLACE 5
;FOLD PROPRIEDADES
MatrizPontos[Pallet_1,Prdt_15CoffeCrisp,5].NumCaixas = 2
MatrizPontos[Pallet_1,Prdt_15CoffeCrisp,5].PickOp = 8
MatrizPontos[Pallet_1,Prdt_15CoffeCrisp,5].ConfGarraOp = 5
MatrizPontos[Pallet_1,Prdt_15CoffeCrisp,5].FechaGarraOp = 0
MatrizPontos[Pallet_1,Prdt_15CoffeCrisp,5].AbreGarraOp = 1
MatrizPontos[Pallet_1,Prdt_15CoffeCrisp,5].SensoresCaixa = 123
MatrizPontos[Pallet_1,Prdt_15CoffeCrisp,5].TravaGarra = True
MatrizPontos[Pallet_1,Prdt_15CoffeCrisp,5].SkipGoHome = False
MatrizPontos[Pallet_1,Prdt_15CoffeCrisp,5].SkipSobeRelAtual = False
MatrizPontos[Pallet_1,Prdt_15CoffeCrisp,5].XApp1Place=P1_15CoffeCrisp_5_App1
MatrizPontos[Pallet_1,Prdt_15CoffeCrisp,5].XApp2Place=P1_15CoffeCrisp_5_App2
MatrizPontos[Pallet_1,Prdt_15CoffeCrisp,5].XPlace=P1_15CoffeCrisp_5_Place
;ENDFOLD
;FOLD OffsetPlace
MatrizPontos[Pallet_1,Prdt_15CoffeCrisp,5].OffsetPlace.X=0
MatrizPontos[Pallet_1,Prdt_15CoffeCrisp,5].OffsetPlace.Y=0
MatrizPontos[Pallet_1,Prdt_15CoffeCrisp,5].OffsetPlace.Z=0
MatrizPontos[Pallet_1,Prdt_15CoffeCrisp,5].OffsetPlace.A=0
MatrizPontos[Pallet_1,Prdt_15CoffeCrisp,5].OffsetPlace.B=0
MatrizPontos[Pallet_1,Prdt_15CoffeCrisp,5].OffsetPlace.C=0
;ENDFOLD
;ENDFOLD

;FOLD PLACE 6
;FOLD PROPRIEDADES
MatrizPontos[Pallet_1,Prdt_15CoffeCrisp,6].NumCaixas = 3
MatrizPontos[Pallet_1,Prdt_15CoffeCrisp,6].PickOp = 8
MatrizPontos[Pallet_1,Prdt_15CoffeCrisp,6].ConfGarraOp = 5
MatrizPontos[Pallet_1,Prdt_15CoffeCrisp,6].FechaGarraOp = 0
MatrizPontos[Pallet_1,Prdt_15CoffeCrisp,6].AbreGarraOp = 0
MatrizPontos[Pallet_1,Prdt_15CoffeCrisp,6].SensoresCaixa = 1234
MatrizPontos[Pallet_1,Prdt_15CoffeCrisp,6].TravaGarra = False
MatrizPontos[Pallet_1,Prdt_15CoffeCrisp,6].SkipGoHome = False
MatrizPontos[Pallet_1,Prdt_15CoffeCrisp,6].SkipSobeRelAtual = False
MatrizPontos[Pallet_1,Prdt_15CoffeCrisp,6].XApp1Place=P1_15CoffeCrisp_6_App1
MatrizPontos[Pallet_1,Prdt_15CoffeCrisp,6].XApp2Place=P1_15CoffeCrisp_6_App2
MatrizPontos[Pallet_1,Prdt_15CoffeCrisp,6].XPlace=P1_15CoffeCrisp_6_Place
;ENDFOLD
;FOLD OffsetPlace
MatrizPontos[Pallet_1,Prdt_15CoffeCrisp,6].OffsetPlace.X=0
MatrizPontos[Pallet_1,Prdt_15CoffeCrisp,6].OffsetPlace.Y=0
MatrizPontos[Pallet_1,Prdt_15CoffeCrisp,6].OffsetPlace.Z=0
MatrizPontos[Pallet_1,Prdt_15CoffeCrisp,6].OffsetPlace.A=0
MatrizPontos[Pallet_1,Prdt_15CoffeCrisp,6].OffsetPlace.B=0
MatrizPontos[Pallet_1,Prdt_15CoffeCrisp,6].OffsetPlace.C=0
;ENDFOLD
;ENDFOLD

;FOLD PLACE 7
;FOLD PROPRIEDADES
MatrizPontos[Pallet_1,Prdt_15CoffeCrisp,7].NumCaixas = 3
MatrizPontos[Pallet_1,Prdt_15CoffeCrisp,7].PickOp = 8
MatrizPontos[Pallet_1,Prdt_15CoffeCrisp,7].ConfGarraOp = 5
MatrizPontos[Pallet_1,Prdt_15CoffeCrisp,7].FechaGarraOp = 0
MatrizPontos[Pallet_1,Prdt_15CoffeCrisp,7].AbreGarraOp = 0
MatrizPontos[Pallet_1,Prdt_15CoffeCrisp,7].SensoresCaixa = 1234
MatrizPontos[Pallet_1,Prdt_15CoffeCrisp,7].TravaGarra = False
MatrizPontos[Pallet_1,Prdt_15CoffeCrisp,7].SkipGoHome = False
MatrizPontos[Pallet_1,Prdt_15CoffeCrisp,7].SkipSobeRelAtual = False
MatrizPontos[Pallet_1,Prdt_15CoffeCrisp,7].XApp1Place=P1_15CoffeCrisp_7_App1
MatrizPontos[Pallet_1,Prdt_15CoffeCrisp,7].XApp2Place=P1_15CoffeCrisp_7_App2
MatrizPontos[Pallet_1,Prdt_15CoffeCrisp,7].XPlace=P1_15CoffeCrisp_7_Place
;ENDFOLD
;FOLD OffsetPlace
MatrizPontos[Pallet_1,Prdt_15CoffeCrisp,7].OffsetPlace.X=0
MatrizPontos[Pallet_1,Prdt_15CoffeCrisp,7].OffsetPlace.Y=0
MatrizPontos[Pallet_1,Prdt_15CoffeCrisp,7].OffsetPlace.Z=0
MatrizPontos[Pallet_1,Prdt_15CoffeCrisp,7].OffsetPlace.A=0
MatrizPontos[Pallet_1,Prdt_15CoffeCrisp,7].OffsetPlace.B=0
MatrizPontos[Pallet_1,Prdt_15CoffeCrisp,7].OffsetPlace.C=0
;ENDFOLD
;ENDFOLD

;ENDFOLD
;FOLD LAYER 2: PLACE 8 ate 14
;FOLD PLACE 8
;FOLD PROPRIEDADES
MatrizPontos[Pallet_1,Prdt_15CoffeCrisp,8].NumCaixas = 1
MatrizPontos[Pallet_1,Prdt_15CoffeCrisp,8].PickOp = 6
MatrizPontos[Pallet_1,Prdt_15CoffeCrisp,8].ConfGarraOp = 5
MatrizPontos[Pallet_1,Prdt_15CoffeCrisp,8].FechaGarraOp = 0
MatrizPontos[Pallet_1,Prdt_15CoffeCrisp,8].AbreGarraOp = 0
MatrizPontos[Pallet_1,Prdt_15CoffeCrisp,8].SensoresCaixa = 1
MatrizPontos[Pallet_1,Prdt_15CoffeCrisp,8].TravaGarra = False
MatrizPontos[Pallet_1,Prdt_15CoffeCrisp,8].SkipGoHome = False
MatrizPontos[Pallet_1,Prdt_15CoffeCrisp,8].SkipSobeRelAtual = False
MatrizPontos[Pallet_1,Prdt_15CoffeCrisp,8].XApp1Place=P1_15CoffeCrisp_8_App1
MatrizPontos[Pallet_1,Prdt_15CoffeCrisp,8].XApp2Place=P1_15CoffeCrisp_8_App2
MatrizPontos[Pallet_1,Prdt_15CoffeCrisp,8].XPlace=P1_15CoffeCrisp_8_Place
;ENDFOLD
;FOLD OffsetPlace
MatrizPontos[Pallet_1,Prdt_15CoffeCrisp,8].OffsetPlace.X=0
MatrizPontos[Pallet_1,Prdt_15CoffeCrisp,8].OffsetPlace.Y=0
MatrizPontos[Pallet_1,Prdt_15CoffeCrisp,8].OffsetPlace.Z=0
MatrizPontos[Pallet_1,Prdt_15CoffeCrisp,8].OffsetPlace.A=0
MatrizPontos[Pallet_1,Prdt_15CoffeCrisp,8].OffsetPlace.B=0
MatrizPontos[Pallet_1,Prdt_15CoffeCrisp,8].OffsetPlace.C=0
;ENDFOLD
;ENDFOLD

;FOLD PLACE 9
;FOLD PROPRIEDADES
MatrizPontos[Pallet_1,Prdt_15CoffeCrisp,9].NumCaixas = 1
MatrizPontos[Pallet_1,Prdt_15CoffeCrisp,9].PickOp = 6
MatrizPontos[Pallet_1,Prdt_15CoffeCrisp,9].ConfGarraOp = 5
MatrizPontos[Pallet_1,Prdt_15CoffeCrisp,9].FechaGarraOp = 0
MatrizPontos[Pallet_1,Prdt_15CoffeCrisp,9].AbreGarraOp = 0
MatrizPontos[Pallet_1,Prdt_15CoffeCrisp,9].SensoresCaixa = 1
MatrizPontos[Pallet_1,Prdt_15CoffeCrisp,9].TravaGarra = False
MatrizPontos[Pallet_1,Prdt_15CoffeCrisp,9].SkipGoHome = False
MatrizPontos[Pallet_1,Prdt_15CoffeCrisp,9].SkipSobeRelAtual = False
MatrizPontos[Pallet_1,Prdt_15CoffeCrisp,9].XApp1Place=P1_15CoffeCrisp_9_App1
MatrizPontos[Pallet_1,Prdt_15CoffeCrisp,9].XApp2Place=P1_15CoffeCrisp_9_App2
MatrizPontos[Pallet_1,Prdt_15CoffeCrisp,9].XPlace=P1_15CoffeCrisp_9_Place
;ENDFOLD
;FOLD OffsetPlace
MatrizPontos[Pallet_1,Prdt_15CoffeCrisp,9].OffsetPlace.X=0
MatrizPontos[Pallet_1,Prdt_15CoffeCrisp,9].OffsetPlace.Y=0
MatrizPontos[Pallet_1,Prdt_15CoffeCrisp,9].OffsetPlace.Z=0
MatrizPontos[Pallet_1,Prdt_15CoffeCrisp,9].OffsetPlace.A=0
MatrizPontos[Pallet_1,Prdt_15CoffeCrisp,9].OffsetPlace.B=0
MatrizPontos[Pallet_1,Prdt_15CoffeCrisp,9].OffsetPlace.C=0
;ENDFOLD
;ENDFOLD

;FOLD PLACE 10
;FOLD PROPRIEDADES
MatrizPontos[Pallet_1,Prdt_15CoffeCrisp,10].NumCaixas = 1
MatrizPontos[Pallet_1,Prdt_15CoffeCrisp,10].PickOp = 6
MatrizPontos[Pallet_1,Prdt_15CoffeCrisp,10].ConfGarraOp = 5
MatrizPontos[Pallet_1,Prdt_15CoffeCrisp,10].FechaGarraOp = 0
MatrizPontos[Pallet_1,Prdt_15CoffeCrisp,10].AbreGarraOp = 0
MatrizPontos[Pallet_1,Prdt_15CoffeCrisp,10].SensoresCaixa = 1
MatrizPontos[Pallet_1,Prdt_15CoffeCrisp,10].TravaGarra = False
MatrizPontos[Pallet_1,Prdt_15CoffeCrisp,10].SkipGoHome = False
MatrizPontos[Pallet_1,Prdt_15CoffeCrisp,10].SkipSobeRelAtual = False
MatrizPontos[Pallet_1,Prdt_15CoffeCrisp,10].XApp1Place=P1_15CoffeCrisp_10_App1
MatrizPontos[Pallet_1,Prdt_15CoffeCrisp,10].XApp2Place=P1_15CoffeCrisp_10_App2
MatrizPontos[Pallet_1,Prdt_15CoffeCrisp,10].XPlace=P1_15CoffeCrisp_10_Place
;ENDFOLD
;FOLD OffsetPlace
MatrizPontos[Pallet_1,Prdt_15CoffeCrisp,10].OffsetPlace.X=0
MatrizPontos[Pallet_1,Prdt_15CoffeCrisp,10].OffsetPlace.Y=0
MatrizPontos[Pallet_1,Prdt_15CoffeCrisp,10].OffsetPlace.Z=0
MatrizPontos[Pallet_1,Prdt_15CoffeCrisp,10].OffsetPlace.A=0
MatrizPontos[Pallet_1,Prdt_15CoffeCrisp,10].OffsetPlace.B=0
MatrizPontos[Pallet_1,Prdt_15CoffeCrisp,10].OffsetPlace.C=0
;ENDFOLD
;ENDFOLD

;FOLD PLACE 11
;FOLD PROPRIEDADES
MatrizPontos[Pallet_1,Prdt_15CoffeCrisp,11].NumCaixas = 2
MatrizPontos[Pallet_1,Prdt_15CoffeCrisp,11].PickOp = 8
MatrizPontos[Pallet_1,Prdt_15CoffeCrisp,11].ConfGarraOp = 5
MatrizPontos[Pallet_1,Prdt_15CoffeCrisp,11].FechaGarraOp = 0
MatrizPontos[Pallet_1,Prdt_15CoffeCrisp,11].AbreGarraOp = 1
MatrizPontos[Pallet_1,Prdt_15CoffeCrisp,11].SensoresCaixa = 123
MatrizPontos[Pallet_1,Prdt_15CoffeCrisp,11].TravaGarra = True
MatrizPontos[Pallet_1,Prdt_15CoffeCrisp,11].SkipGoHome = False
MatrizPontos[Pallet_1,Prdt_15CoffeCrisp,11].SkipSobeRelAtual = False
MatrizPontos[Pallet_1,Prdt_15CoffeCrisp,11].XApp1Place=P1_15CoffeCrisp_11_App1
MatrizPontos[Pallet_1,Prdt_15CoffeCrisp,11].XApp2Place=P1_15CoffeCrisp_11_App2
MatrizPontos[Pallet_1,Prdt_15CoffeCrisp,11].XPlace=P1_15CoffeCrisp_11_Place
;ENDFOLD
;FOLD OffsetPlace
MatrizPontos[Pallet_1,Prdt_15CoffeCrisp,11].OffsetPlace.X=0
MatrizPontos[Pallet_1,Prdt_15CoffeCrisp,11].OffsetPlace.Y=0
MatrizPontos[Pallet_1,Prdt_15CoffeCrisp,11].OffsetPlace.Z=0
MatrizPontos[Pallet_1,Prdt_15CoffeCrisp,11].OffsetPlace.A=0
MatrizPontos[Pallet_1,Prdt_15CoffeCrisp,11].OffsetPlace.B=0
MatrizPontos[Pallet_1,Prdt_15CoffeCrisp,11].OffsetPlace.C=0
;ENDFOLD
;ENDFOLD

;FOLD PLACE 12
;FOLD PROPRIEDADES
MatrizPontos[Pallet_1,Prdt_15CoffeCrisp,12].NumCaixas = 2
MatrizPontos[Pallet_1,Prdt_15CoffeCrisp,12].PickOp = 8
MatrizPontos[Pallet_1,Prdt_15CoffeCrisp,12].ConfGarraOp = 5
MatrizPontos[Pallet_1,Prdt_15CoffeCrisp,12].FechaGarraOp = 0
MatrizPontos[Pallet_1,Prdt_15CoffeCrisp,12].AbreGarraOp = 1
MatrizPontos[Pallet_1,Prdt_15CoffeCrisp,12].SensoresCaixa = 123
MatrizPontos[Pallet_1,Prdt_15CoffeCrisp,12].TravaGarra = True
MatrizPontos[Pallet_1,Prdt_15CoffeCrisp,12].SkipGoHome = False
MatrizPontos[Pallet_1,Prdt_15CoffeCrisp,12].SkipSobeRelAtual = False
MatrizPontos[Pallet_1,Prdt_15CoffeCrisp,12].XApp1Place=P1_15CoffeCrisp_12_App1
MatrizPontos[Pallet_1,Prdt_15CoffeCrisp,12].XApp2Place=P1_15CoffeCrisp_12_App2
MatrizPontos[Pallet_1,Prdt_15CoffeCrisp,12].XPlace=P1_15CoffeCrisp_12_Place
;ENDFOLD
;FOLD OffsetPlace
MatrizPontos[Pallet_1,Prdt_15CoffeCrisp,12].OffsetPlace.X=0
MatrizPontos[Pallet_1,Prdt_15CoffeCrisp,12].OffsetPlace.Y=0
MatrizPontos[Pallet_1,Prdt_15CoffeCrisp,12].OffsetPlace.Z=0
MatrizPontos[Pallet_1,Prdt_15CoffeCrisp,12].OffsetPlace.A=0
MatrizPontos[Pallet_1,Prdt_15CoffeCrisp,12].OffsetPlace.B=0
MatrizPontos[Pallet_1,Prdt_15CoffeCrisp,12].OffsetPlace.C=0
;ENDFOLD
;ENDFOLD

;FOLD PLACE 13
;FOLD PROPRIEDADES
MatrizPontos[Pallet_1,Prdt_15CoffeCrisp,13].NumCaixas = 3
MatrizPontos[Pallet_1,Prdt_15CoffeCrisp,13].PickOp = 6
MatrizPontos[Pallet_1,Prdt_15CoffeCrisp,13].ConfGarraOp = 5
MatrizPontos[Pallet_1,Prdt_15CoffeCrisp,13].FechaGarraOp = 0
MatrizPontos[Pallet_1,Prdt_15CoffeCrisp,13].AbreGarraOp = 1
MatrizPontos[Pallet_1,Prdt_15CoffeCrisp,13].SensoresCaixa = 1234
MatrizPontos[Pallet_1,Prdt_15CoffeCrisp,13].TravaGarra = True
MatrizPontos[Pallet_1,Prdt_15CoffeCrisp,13].SkipGoHome = False
MatrizPontos[Pallet_1,Prdt_15CoffeCrisp,13].SkipSobeRelAtual = False
MatrizPontos[Pallet_1,Prdt_15CoffeCrisp,13].XApp1Place=P1_15CoffeCrisp_13_App1
MatrizPontos[Pallet_1,Prdt_15CoffeCrisp,13].XApp2Place=P1_15CoffeCrisp_13_App2
MatrizPontos[Pallet_1,Prdt_15CoffeCrisp,13].XPlace=P1_15CoffeCrisp_13_Place
;ENDFOLD
;FOLD OffsetPlace
MatrizPontos[Pallet_1,Prdt_15CoffeCrisp,13].OffsetPlace.X=0
MatrizPontos[Pallet_1,Prdt_15CoffeCrisp,13].OffsetPlace.Y=0
MatrizPontos[Pallet_1,Prdt_15CoffeCrisp,13].OffsetPlace.Z=0
MatrizPontos[Pallet_1,Prdt_15CoffeCrisp,13].OffsetPlace.A=0
MatrizPontos[Pallet_1,Prdt_15CoffeCrisp,13].OffsetPlace.B=0
MatrizPontos[Pallet_1,Prdt_15CoffeCrisp,13].OffsetPlace.C=0
;ENDFOLD
;ENDFOLD

